FUNCTION_BLOCK FB_Heating_System_Manager
  VAR_INPUT
    VI_System_Mode : E_System_Operating_Mode;
    VI_System_Time_MS : UDINT;
    VI_Current_TOD : TOD;
    VI_IsActivePLC : BOOL;
    VI_Outdoor_Temp : REAL;
    VI_Config : ST_Heating_Config;
    VI_Tariff : ST_Tariff_Config;
    VI_Current_Hour : UINT;
    VI_Boiler_Stop : BOOL;
    VI_DHW_Heating_Demand : BOOL;
    VI_DHW_Target_Temp : REAL;
    VI_Current_Scenario : E_SCENARIO_TYPE;
    VI_Emergency_Stop : BOOL;
    VI_Gas_Safety_Stop : BOOL;
    VI_Boiler_Error_Status : ARRAY[1..GVL_CONSTANTS.C_MAX_BOILERS] OF BOOL;
    VI_Boiler_OT_Online : ARRAY[1..GVL_CONSTANTS.C_MAX_BOILERS] OF BOOL;
    VI_Boiler_Modulation : ARRAY[1..GVL_CONSTANTS.C_MAX_BOILERS] OF REAL;
  END_VAR
  VAR_OUTPUT
    VO_Manifold_Valves : ARRAY[1..GVL_CONSTANTS.C_MAX_MANIFOLDS] OF REAL;
    VO_Manifold_Pumps : ARRAY[1..GVL_CONSTANTS.C_MAX_MANIFOLDS] OF BOOL;
    VO_Zone_Valves : ARRAY[1..GVL_CONSTANTS.C_MAX_HEATING_CIRCUITS] OF BOOL;
    VO_Boiler_OT_Enable : ARRAY[1..GVL_CONSTANTS.C_MAX_BOILERS] OF BOOL;
    VO_Boiler_OT_Setpoint : ARRAY[1..GVL_CONSTANTS.C_MAX_BOILERS] OF REAL;
    VO_Backup_Circulation_Pump : BOOL;
    VO_Electric_Heater_Enable : BOOL;
    VO_Freeze_Risk_Status : BOOL;
    VO_Status : ARRAY[1..GVL_CONSTANTS.C_MAX_MANIFOLDS] OF ST_Manifold_Status;
    VO_Boiler_Status : ARRAY[1..GVL_CONSTANTS.C_MAX_BOILERS] OF ST_Boiler_Status;
  END_VAR
  VAR_IN_OUT
    VI_Floor_Temps : ARRAY[1..GVL_CONSTANTS.C_MAX_HEATING_CIRCUITS] OF REAL;
    VI_Room_Temps : ARRAY[1..GVL_CONSTANTS.C_MAX_CLIMATE_ZONES] OF REAL;
    VI_Manifold_Pressures : ARRAY[1..GVL_CONSTANTS.C_MAX_MANIFOLDS] OF REAL;
    VI_Manifold_Currents : ARRAY[1..GVL_CONSTANTS.C_MAX_MANIFOLDS] OF REAL;
    VI_Manifold_Temps_Supply : ARRAY[1..GVL_CONSTANTS.C_MAX_MANIFOLDS] OF REAL;
    VI_Manifold_Temps_Return : ARRAY[1..GVL_CONSTANTS.C_MAX_MANIFOLDS] OF REAL;
    VI_Boiler_Flame_Status : ARRAY[1..GVL_CONSTANTS.C_MAX_BOILERS] OF BOOL;
    VI_Zone_Configs : ARRAY[1..GVL_CONSTANTS.C_MAX_HEATING_CIRCUITS] OF ST_FloorHeating_Circuit_Config;
    VI_Rule_Actions : ARRAY[1..GVL_CONSTANTS.C_MAX_RULES] OF ST_Rule_Action;
    VI_IO_Modules_Online : ARRAY[1..GVL_CONSTANTS.C_MAX_MODULES] OF BOOL;
    VI_Scenario_Configs : ARRAY[1..GVL_CONSTANTS.C_MAX_SCENARIOS] OF ST_Scenario_Config;
    VI_Manifold_End_Switches : ARRAY[1..GVL_CONSTANTS.C_MAX_MANIFOLDS] OF BOOL;
    VI_Valve_Test_Config : ARRAY[1..GVL_CONSTANTS.C_MAX_MANIFOLDS] OF ST_Valve_Test_Config;
  END_VAR
  VAR
    fbHeatingV2Staging : FB_Heating_V2_Staging_DRAFT;
    L_Heating_V2_Command_Shadow : ST_Heating_Command_V2;
    L_Heating_V2_State_Shadow : ST_Heating_State_V2;
    L_Heating_V2_Shadow_Diff_Found : BOOL;
    L_Heating_V2_Switch_Enabled : BOOL;
    L_Heating_V2_Path_Ready : BOOL;
    L_Heating_Using_Legacy_Fallback : BOOL;
    L_PID_Valves : ARRAY[1..GVL_CONSTANTS.C_MAX_MANIFOLDS] OF FB_PID_Controller;
    L_PID_Timer : ARRAY[1..GVL_CONSTANTS.C_MAX_MANIFOLDS] OF FB_System_Timer;
    L_Floor_Controllers : ARRAY[1..GVL_CONSTANTS.C_MAX_HEATING_CIRCUITS] OF FB_FloorHeating_Controller;
    L_Last_Boiler_Rotation : UDINT;
    L_Lead_Boiler : BYTE := 1;
    L_i : INT;
    L_Zone_Config : ST_FloorHeating_Circuit_Config;
    L_j : INT;
    L_Target_Supply_Temp : REAL;
    L_Demand_Power : REAL;
    L_Any_Zone_Active : ARRAY[1..GVL_CONSTANTS.C_MAX_MANIFOLDS] OF BOOL;
    L_Current_Temp : REAL;
    L_Sensor_Error : BOOL;
    L_Prev_Scenario : E_SCENARIO_TYPE;
    L_Scenario_Adjust : REAL;
    L_Target_Scenario_Adjust : REAL;
    L_Transition_Temp : FB_Scenario_Transition_Controller;
    L_Overheat_Timer : ARRAY[1..GVL_CONSTANTS.C_MAX_HEATING_CIRCUITS] OF FB_System_Timer;
    L_Pump_Run_Timer : ARRAY[1..GVL_CONSTANTS.C_MAX_MANIFOLDS] OF FB_System_Timer;
    L_Pump_Pause_Timer : ARRAY[1..GVL_CONSTANTS.C_MAX_MANIFOLDS] OF FB_System_Timer;
    L_Pump_In_Pause : ARRAY[1..GVL_CONSTANTS.C_MAX_MANIFOLDS] OF BOOL;
    L_Last_Scan_Time : UDINT;
    L_Scan_Time_Init : BOOL := FALSE;
    L_Lifespan_S : REAL := 50000.0 * 3600.0;
    L_Delta_MS : UDINT;
    L_Pump_Diag : ARRAY[1..GVL_CONSTANTS.C_MAX_MANIFOLDS] OF FB_Device_Predictive_Diag;
    L_Boiler_Life : ARRAY[1..GVL_CONSTANTS.C_MAX_BOILERS] OF FB_Lifetime_Predictor;
    fbFloorTempValidator : ARRAY[1..GVL_CONSTANTS.C_MAX_HEATING_CIRCUITS] OF FB_Analog_Validator;
    fbRoomTempValidator : ARRAY[1..GVL_CONSTANTS.C_MAX_CLIMATE_ZONES] OF FB_Analog_Validator;
    fbValveTestManager : FB_Valve_Test_Manager;
    fbBoilerCascade : FB_Boiler_Cascade_Manager;
    fbBoilerOpenTherm : FB_Boiler_OpenTherm_Interface;
    L_IO_Failsafe_Active : BOOL;
    L_Freeze_Mode_Active : BOOL;
    L_Freeze_Target_Supply : REAL;
    L_Delta_T : REAL;
    L_Min_Supply_Temp : REAL;
    L_Boiler_OT_Command_Valid : ARRAY[1..GVL_CONSTANTS.C_MAX_BOILERS] OF BOOL;
    L_Boiler_Request_Enable : ARRAY[1..GVL_CONSTANTS.C_MAX_BOILERS] OF BOOL;
    L_Boiler_Request_Setpoint : ARRAY[1..GVL_CONSTANTS.C_MAX_BOILERS] OF REAL;
    L_Policy_Normal : BOOL;
    L_Policy_Safe_Stop : BOOL;
    L_Policy_Degraded : BOOL;
    L_Policy_Freeze_Protection : BOOL;
    L_Any_Sensor_Error : BOOL;
    L_Any_Subsystem_Degraded : BOOL;
  END_VAR

      // ==============================================================================
// Блок управления системой отопления (Heating System Manager)
// Назначение:
// - Управление контурами теплого пола (открытие/закрытие клапанов).
// - Управление насосами коллекторов и смесительными узлами.
// - Управление каскадом котлов (ротация, расчет ресурса).
// - Защита от перегрева и замерзания.
// - Интеграция с Rule Engine.
// ==============================================================================





// ========================================
// Heating policy layer (phase2)
// ========================================
L_Policy_Normal := (VI_System_Mode = E_System_Operating_Mode.MODE_NORMAL);
L_Policy_Safe_Stop := (VI_System_Mode = E_System_Operating_Mode.MODE_SAFE_STOP);
L_Policy_Degraded := (VI_System_Mode = E_System_Operating_Mode.MODE_DEGRADED);
L_Policy_Freeze_Protection := (VI_System_Mode = E_System_Operating_Mode.MODE_FREEZE_PROTECTION);

// ========================================
// Heating freeze policy activation
// ========================================
IF L_Policy_Freeze_Protection THEN
    L_Freeze_Mode_Active := TRUE;
END_IF;

// 0. Агрегация деградации для system mode
GVL_STATE.G_Heating_IO_Fault := FALSE;
GVL_STATE.G_Heating_Sensor_Fault := FALSE;
GVL_STATE.G_Heating_Subsystem_Degraded := FALSE;
L_Any_Sensor_Error := FALSE;
L_Any_Subsystem_Degraded := FALSE;
L_Heating_V2_Shadow_Diff_Found := FALSE;
L_Heating_V2_Switch_Enabled := TRUE;
L_Heating_V2_Path_Ready := FALSE;
L_Heating_Using_Legacy_Fallback := TRUE;

// 0. Аварийный стоп от подсистемы безопасности
VO_Backup_Circulation_Pump := FALSE;
VO_Electric_Heater_Enable := FALSE;
VO_Freeze_Risk_Status := FALSE;

IF VI_Gas_Safety_Stop THEN
    L_Freeze_Mode_Active := (VI_Outdoor_Temp < -5.0);
    FOR L_i := 1 TO GVL_CONSTANTS.C_MAX_HEATING_CIRCUITS DO
        IF VI_Floor_Temps[L_i] < 7.0 THEN
            L_Freeze_Mode_Active := TRUE;
        END_IF;
        VO_Zone_Valves[L_i] := FALSE;
    END_FOR;

    FOR L_i := 1 TO GVL_CONSTANTS.C_MAX_MANIFOLDS DO
        VO_Manifold_Pumps[L_i] := FALSE;
        VO_Manifold_Valves[L_i] := 0.0;
    END_FOR;

    FOR L_i := 1 TO GVL_CONSTANTS.C_MAX_BOILERS DO
        VO_Boiler_OT_Enable[L_i] := FALSE;
        VO_Boiler_OT_Setpoint[L_i] := 0.0;
        VO_Boiler_Status[L_i].Warning := FALSE;
        VO_Boiler_Status[L_i].Error := TRUE;
    END_FOR;

    IF L_Freeze_Mode_Active THEN
        VO_Backup_Circulation_Pump := TRUE;
        L_Freeze_Target_Supply := LIMIT(20.0, VI_Config.Freeze_Threshold + 2.0, 35.0);
        L_Min_Supply_Temp := 1000.0;
        FOR L_i := 1 TO GVL_CONSTANTS.C_MAX_MANIFOLDS DO
            IF VI_Manifold_Temps_Supply[L_i] < L_Min_Supply_Temp THEN
                L_Min_Supply_Temp := VI_Manifold_Temps_Supply[L_i];
            END_IF;
        END_FOR;
        IF L_Min_Supply_Temp > 900.0 THEN
            L_Min_Supply_Temp := 0.0;
        END_IF;

        IF L_Min_Supply_Temp < (L_Freeze_Target_Supply - 1.0) THEN
            VO_Electric_Heater_Enable := TRUE;
        ELSIF L_Min_Supply_Temp > (L_Freeze_Target_Supply + 1.0) THEN
            VO_Electric_Heater_Enable := FALSE;
        END_IF;

        // При защёлкнутой газовой аварии оператор должен видеть, что система живёт в деградированном anti-freeze режиме.
        VO_Freeze_Risk_Status := TRUE;
    END_IF;

    RETURN;
END_IF;

IF VI_Emergency_Stop OR L_Policy_Safe_Stop THEN
    FOR L_i := 1 TO GVL_CONSTANTS.C_MAX_HEATING_CIRCUITS DO
        VO_Zone_Valves[L_i] := FALSE;
    END_FOR;

    FOR L_i := 1 TO GVL_CONSTANTS.C_MAX_MANIFOLDS DO
        VO_Manifold_Pumps[L_i] := FALSE;
        VO_Manifold_Valves[L_i] := 0.0;
    END_FOR;

    FOR L_i := 1 TO GVL_CONSTANTS.C_MAX_BOILERS DO
        VO_Boiler_OT_Enable[L_i] := FALSE;
        VO_Boiler_OT_Setpoint[L_i] := 0.0;
        VO_Boiler_Status[L_i].Warning := FALSE;
        VO_Boiler_Status[L_i].Error := TRUE;
    END_FOR;

    RETURN;
END_IF;

// 1. Проверка связи с модулями ввода-вывода (ТЗ 2.0)
L_IO_Failsafe_Active := FALSE;
FOR L_i := 1 TO GVL_CONSTANTS.C_MAX_MODULES DO
    IF NOT VI_IO_Modules_Online[L_i] THEN
        L_IO_Failsafe_Active := TRUE;
        GVL_STATE.G_Heating_IO_Fault := TRUE;
GVL_STATE.G_Heating_Subsystem_Degraded := TRUE;
        EXIT;
    END_IF;
END_FOR;

IF L_IO_Failsafe_Active THEN
    // Fail-safe: закрываем зональные клапаны, чтобы не разгонять неконтролируемые контуры,
    // но при риске замерзания сохраняем минимальную циркуляцию и минимальную теплогенерацию.
    L_Freeze_Mode_Active := (VI_Outdoor_Temp < -5.0);

    FOR L_j := 1 TO GVL_CONSTANTS.C_MAX_HEATING_CIRCUITS DO
        IF VI_Floor_Temps[L_j] < 7.0 THEN
            L_Freeze_Mode_Active := TRUE;
        END_IF;
        VO_Zone_Valves[L_j] := FALSE;
    END_FOR;

    IF L_Freeze_Mode_Active THEN
        L_Freeze_Target_Supply := LIMIT(20.0, VI_Config.Freeze_Threshold + 2.0, 35.0);
    ELSE
        L_Freeze_Target_Supply := 0.0;
    END_IF;

    FOR L_j := 1 TO GVL_CONSTANTS.C_MAX_MANIFOLDS DO
        IF L_Freeze_Mode_Active THEN
            VO_Manifold_Pumps[L_j] := TRUE;
            VO_Manifold_Valves[L_j] := 35.0;
        ELSE
            VO_Manifold_Pumps[L_j] := FALSE;
            VO_Manifold_Valves[L_j] := 0.0;
        END_IF;
    END_FOR;

    // В аварийном I/O режиме напрямую формируем только legacy request-мirror.
    // Реальные физические команды всё равно будут интерпретированы transport-слоем выше по архитектуре.
    FOR L_j := 1 TO GVL_CONSTANTS.C_MAX_BOILERS DO
        VO_Boiler_OT_Enable[L_j] := FALSE;
        VO_Boiler_OT_Setpoint[L_j] := 0.0;
    END_FOR;

    IF L_Freeze_Mode_Active THEN
        // В fail-safe используем только ведущий аварийный вариант: котёл №1 на минимальной уставке.
        IF VI_Boiler_OT_Online[1] AND NOT VI_Boiler_Error_Status[1] THEN
            VO_Boiler_OT_Enable[1] := TRUE;
            VO_Boiler_OT_Setpoint[1] := L_Freeze_Target_Supply;
        END_IF;
    END_IF;

    RETURN;
END_IF;

// 2. Расчет целевой температуры подачи теплоносителя (Погодозависимая автоматика ТЗ 2.3)
L_Target_Supply_Temp := 35.0; // Базовая уставка
IF VI_Config.Weather_Comp_Enabled AND VI_Outdoor_Temp < 15.0 THEN
    // Коррекция по уличному датчику с использованием коэффициента кривой
    L_Target_Supply_Temp := L_Target_Supply_Temp + (15.0 - VI_Outdoor_Temp) * VI_Config.Weather_Coef;
END_IF;
L_Target_Supply_Temp := LIMIT(20.0, L_Target_Supply_Temp, 45.0); // Ограничение диапазона для теплого пола

IF L_Policy_Degraded THEN
    IF L_Target_Supply_Temp > 35.0 THEN
        L_Target_Supply_Temp := 35.0;
    END_IF;
END_IF;

// Плавный переход уставки по сценарию
IF VI_Current_Scenario >= 1 AND VI_Current_Scenario <= GVL_CONSTANTS.C_MAX_SCENARIOS THEN
    L_Target_Scenario_Adjust := VI_Scenario_Configs[VI_Current_Scenario].floor_heating_adjust_celsius;
ELSE
    L_Target_Scenario_Adjust := 0.0;
END_IF;

IF VI_Current_Scenario <> L_Prev_Scenario THEN
    L_Transition_Temp(
        VI_System_Time := VI_System_Time_MS,
        VI_Start_Time := VI_System_Time_MS,
        VI_Duration := 300000, // 5 минут на плавное изменение температуры
        VI_Start_Value := L_Scenario_Adjust,
        VI_End_Value := L_Target_Scenario_Adjust
    );
    L_Prev_Scenario := VI_Current_Scenario;
ELSE
    L_Transition_Temp(
        VI_System_Time := VI_System_Time_MS,
        VI_Start_Time := L_Transition_Temp.VI_Start_Time,
        VI_Duration := L_Transition_Temp.VI_Duration,
        VI_Start_Value := L_Transition_Temp.VI_Start_Value,
        VI_End_Value := L_Target_Scenario_Adjust
    );
END_IF;
L_Scenario_Adjust := L_Transition_Temp.VO_Current_Value;

// ТЗ 2.4: Защита от замерзания по температуре пола < 7°C или наружной < -5°C
L_Freeze_Mode_Active := L_Policy_Freeze_Protection OR (VI_Outdoor_Temp < -5.0);
IF NOT L_Freeze_Mode_Active THEN
    FOR L_i := 1 TO GVL_CONSTANTS.C_MAX_HEATING_CIRCUITS DO
        IF VI_Floor_Temps[L_i] < 7.0 THEN
            L_Freeze_Mode_Active := TRUE;
            EXIT;
        END_IF;
    END_FOR;
END_IF;

IF L_Freeze_Mode_Active THEN
    L_Freeze_Target_Supply := LIMIT(20.0, VI_Config.Freeze_Threshold + 2.0, 45.0);
    IF L_Target_Supply_Temp < L_Freeze_Target_Supply THEN
        L_Target_Supply_Temp := L_Freeze_Target_Supply;
    END_IF;
END_IF;

// 2. Индивидуальное управление зонами отопления (ТЗ 1.1, 2.5)
FOR L_i := 1 TO GVL_CONSTANTS.C_MAX_HEATING_CIRCUITS DO
    fbFloorTempValidator[L_i](
        VI_Value := VI_Floor_Temps[L_i],
        VI_Min_Valid := -40.0,
        VI_Max_Valid := 120.0,
        VI_Fallback_Mode := 0
    );
    
    L_Climate_Zone_ID := VI_Zone_Configs[L_i].zone;
    IF L_Climate_Zone_ID >= 1 AND L_Climate_Zone_ID <= GVL_CONSTANTS.C_MAX_CLIMATE_ZONES THEN
        fbRoomTempValidator[L_Climate_Zone_ID](
        VI_Value := VI_Room_Temps[L_Climate_Zone_ID],
        VI_Min_Valid := -40.0,
        VI_Max_Valid := 120.0,
        VI_Fallback_Mode := 0
        );
    END_IF;

    // Контроль перегрева стяжки (защита напольного покрытия)
    L_Overheat_Timer[L_i](IN := fbFloorTempValidator[L_i].VO_Value > VI_Config.Overheat_Threshold, PT := T#60s, VI_System_Time_MS := VI_System_Time_MS);
    
    // Выбор датчика температуры с автоматическим переключением при неисправности
    L_Current_Temp := 0.0;
    L_Sensor_Error := FALSE;
    
    IF VI_Zone_Configs[L_i].control_type = 1 OR VI_Zone_Configs[L_i].control_type = 2 THEN
        // Основной: по воздуху
        IF NOT fbRoomTempValidator[L_Climate_Zone_ID].VO_Error THEN
            L_Current_Temp := fbRoomTempValidator[L_Climate_Zone_ID].VO_Value;
        ELSIF NOT fbFloorTempValidator[L_i].VO_Error THEN
            L_Current_Temp := fbFloorTempValidator[L_i].VO_Value; // Резервный: по полу
        ELSE
            L_Sensor_Error := TRUE;
        END_IF;
    ELSE
        // Основной: по полу
        IF NOT fbFloorTempValidator[L_i].VO_Error THEN
            L_Current_Temp := fbFloorTempValidator[L_i].VO_Value;
        ELSIF NOT fbRoomTempValidator[L_Climate_Zone_ID].VO_Error THEN
            L_Current_Temp := fbRoomTempValidator[L_Climate_Zone_ID].VO_Value; // Резервный: по воздуху
        ELSE
            L_Sensor_Error := TRUE;
        END_IF;
    END_IF;

    IF L_Sensor_Error THEN
        L_Any_Sensor_Error := TRUE;
        VO_Zone_Valves[L_i] := FALSE; // Безопасное состояние при ошибке обоих датчиков
    ELSE
        // ПИД-регулирование и ШИМ для каждой зоны
        // Применяем плавную корректировку уставки от сценария
        L_Zone_Config := VI_Zone_Configs[L_i];
        L_Zone_Config.design_temp := L_Zone_Config.design_temp + L_Scenario_Adjust;
        L_Floor_Controllers[L_i](
            VI_Current_Temp := L_Current_Temp,
            VI_Config := L_Zone_Config,
            VI_Tariff := VI_Tariff,
            VI_Current_Hour := VI_Current_Hour,
            VI_IsActivePLC := VI_IsActivePLC,
            VI_System_Time_MS := VI_System_Time_MS,
            VO_Valve_Bool => VO_Zone_Valves[L_i]
        );
    END_IF;
    
    // Принудительное закрытие клапана при перегреве пола (ТЗ 2.5)
    IF L_Overheat_Timer[L_i].Q THEN
        VO_Zone_Valves[L_i] := FALSE;
    END_IF;
    
    // Обработка действий от Rule Engine (ТЗ 13.0)
    FOR L_j := 1 TO GVL_CONSTANTS.C_MAX_RULES DO
        IF VI_Rule_Actions[L_j].Active AND VI_Rule_Actions[L_j].Target_ID = L_i THEN
            IF VI_Rule_Actions[L_j].Action_Type = E_Rule_Action_Type.ACTION_SET_FLOOR_HEATING THEN
                VO_Zone_Valves[L_i] := (VI_Rule_Actions[L_j].Value > 0.5);
            END_IF;
        END_IF;
    END_FOR;
END_FOR;

GVL_STATE.G_Heating_Sensor_Fault := L_Any_Sensor_Error;

// 3. Определение потребности в работе коллекторных насосов
FOR L_i := 1 TO GVL_CONSTANTS.C_MAX_MANIFOLDS DO
    L_Any_Zone_Active[L_i] := FALSE;
END_FOR;

FOR L_i := 1 TO GVL_CONSTANTS.C_MAX_HEATING_CIRCUITS DO
    IF VO_Zone_Valves[L_i] THEN
        L_j := VI_Zone_Configs[L_i].manifold_id;
        IF L_j >= 1 AND L_j <= GVL_CONSTANTS.C_MAX_MANIFOLDS THEN
            L_Any_Zone_Active[L_j] := TRUE;
        END_IF;
    END_IF;
END_FOR;

// 4. Управление смесительными узлами коллекторов (ТЗ 2.6, 12.2)
FOR L_i := 1 TO GVL_CONSTANTS.C_MAX_MANIFOLDS DO
    // ПИД-регулирование трехходового клапана для поддержания стабильной температуры подачи
    // Вызываем ПИД регулятор каждую секунду
    L_PID_Timer[L_i](IN := TRUE, PT := T#1s, VI_System_Time_MS := VI_System_Time_MS);
    IF L_PID_Timer[L_i].Q THEN
        L_PID_Timer[L_i](IN := FALSE, PT := T#1s, VI_System_Time_MS := VI_System_Time_MS); // Сброс таймера
        L_PID_Timer[L_i](IN := TRUE, PT := T#1s, VI_System_Time_MS := VI_System_Time_MS); // Перезапуск
        
        L_PID_Valves[L_i](
            VI_SetPoint := L_Target_Supply_Temp,
            VI_ProcessValue := VI_Manifold_Temps_Supply[L_i],
            VI_Kp := 2.0, VI_Tn := 120.0, VI_Tv := 0.0,
            VI_Y_Min := 0.0, VI_Y_Max := 100.0, VI_Cycle_Time_S := 1.0,
            VO_Output => VO_Manifold_Valves[L_i]
        );
    END_IF;

    // ТЗ 2.6: Реализация обязательной паузы насоса (защита от закисания и перегрева при 72ч работе)
    L_Pump_Run_Timer[L_i](IN := VO_Manifold_Pumps[L_i] AND NOT L_Pump_In_Pause[L_i], PT := T#72h, VI_System_Time_MS := VI_System_Time_MS);
    IF L_Pump_Run_Timer[L_i].Q THEN L_Pump_In_Pause[L_i] := TRUE; END_IF;
    
    L_Pump_Pause_Timer[L_i](IN := L_Pump_In_Pause[L_i], PT := T#1h, VI_System_Time_MS := VI_System_Time_MS);
    IF L_Pump_Pause_Timer[L_i].Q THEN L_Pump_In_Pause[L_i] := FALSE; END_IF;

    // Включение насоса при наличии запроса от зон и отсутствии сервисной паузы
    // Приоритет ГВС: если есть запрос от ГВС, отключаем насосы отопления и закрываем клапаны
    IF VI_DHW_Heating_Demand THEN
        VO_Manifold_Pumps[L_i] := FALSE;
        VO_Manifold_Valves[L_i] := 0.0; // Принудительно закрываем смесительный клапан
    ELSE
        VO_Manifold_Pumps[L_i] := VI_IsActivePLC AND L_Any_Zone_Active[L_i] AND NOT L_Pump_In_Pause[L_i];
    END_IF;

    // Защита от замерзания системы (ТЗ 2.4)
        IF L_Freeze_Mode_Active THEN
            VO_Manifold_Pumps[L_i] := TRUE;
            IF VO_Manifold_Valves[L_i] < 35.0 THEN
                VO_Manifold_Valves[L_i] := 35.0;
            END_IF;
        END_IF;

        // Сбор диагностических данных для визуализации на HMI
    VO_Status[L_i].Pump_On := VO_Manifold_Pumps[L_i];
    VO_Status[L_i].Pump_Current := VI_Manifold_Currents[L_i];
    VO_Status[L_i].Pressure := VI_Manifold_Pressures[L_i];
    VO_Status[L_i].Temp_Supply := VI_Manifold_Temps_Supply[L_i];
    VO_Status[L_i].Temp_Return := VI_Manifold_Temps_Return[L_i];
    VO_Status[L_i].Valve_Pos := VO_Manifold_Valves[L_i];
    
    // Предиктивная диагностика насоса
    L_Pump_Diag[L_i](
        VI_Current_Value := VI_Manifold_Currents[L_i],
        VI_Nominal_Value := 0.55, // Номинальный ток насоса по ТЗ: середина диапазона 0.3..0.8 А
        VI_Is_Running := VO_Manifold_Pumps[L_i],
        VI_Reset_Stats := FALSE,
        VI_System_Time_MS := VI_System_Time_MS,
        VIO_Health_Data := VO_Status[L_i].Health
    );
    
    // Автоматический контроль рабочих параметров (ток / давление / ΔT)
        IF VO_Manifold_Pumps[L_i] THEN
            L_Delta_T := VI_Manifold_Temps_Supply[L_i] - VI_Manifold_Temps_Return[L_i];

            // Контроль тока насоса:
            // Приоритет ошибок:
            // 1. Насос/ток
            // 2. Давление
            // 3. ΔT
            VO_Status[L_i].Error := FALSE;
            VO_Status[L_i].Error_ID := 0;

            IF VI_Manifold_Currents[L_i] <= 0.01 THEN
                VO_Status[L_i].Error := TRUE;
                VO_Status[L_i].Error_ID := GVL_CONFIG.ERR_PUMP_NO_CURRENT;
            ELSIF VI_Manifold_Currents[L_i] < 0.3 THEN
                VO_Status[L_i].Error := TRUE;
                VO_Status[L_i].Error_ID := GVL_CONFIG.ERR_PUMP_UNDERCURRENT;
            ELSIF VI_Manifold_Currents[L_i] > 1.5 THEN
                VO_Status[L_i].Error := TRUE;
                VO_Status[L_i].Error_ID := GVL_CONFIG.ERR_PUMP_OVERCURRENT;
            END_IF;

            // Проверка давления в системе (норма 1.5 - 2.5 бар)
            IF (NOT VO_Status[L_i].Error) AND (VI_Manifold_Pressures[L_i] < 1.5 OR VI_Manifold_Pressures[L_i] > 2.5) THEN
                VO_Status[L_i].Error := TRUE;
                VO_Status[L_i].Error_ID := GVL_CONFIG.ERR_PRESSURE_OUT_OF_RANGE;
            END_IF;

            // Проверка эффективности теплообмена (ΔT 5..10°C норма)
            IF NOT VO_Status[L_i].Error THEN
                IF L_Delta_T < 5.0 THEN
                    VO_Status[L_i].Error := TRUE;
                    VO_Status[L_i].Error_ID := GVL_CONFIG.ERR_DELTA_T_LOW;
                ELSIF L_Delta_T > 10.0 THEN
                    VO_Status[L_i].Error := TRUE;
                    VO_Status[L_i].Error_ID := GVL_CONFIG.ERR_DELTA_T_HIGH;
                END_IF;
            END_IF;
        END_IF;

        // ТЗ 12.2: Еженедельное тестирование запорной арматуры (предотвращение закисания)
    // Выполняется менеджером fbValveTestManager
END_FOR;

fbValveTestManager(
    VI_System_Time_MS := VI_System_Time_MS,
    VI_IsActivePLC := VI_IsActivePLC,
    VI_Valve_Currents := VI_Manifold_Currents,
    VI_Valve_End_Switches := VI_Manifold_End_Switches,
    VI_Config := VI_Valve_Test_Config
);

IF fbValveTestManager.VO_Test_Active THEN
    L_i := fbValveTestManager.VO_Current_Valve;
    IF L_i >= 1 AND L_i <= GVL_CONSTANTS.C_MAX_MANIFOLDS THEN
        IF fbValveTestManager.VO_Valve_Cmd[L_i] THEN
            VO_Manifold_Valves[L_i] := 100.0;
        ELSE
            VO_Manifold_Valves[L_i] := 0.0;
        END_IF;
        VO_Manifold_Pumps[L_i] := FALSE; // Отключаем насос при тестировании клапана
    END_IF;
END_IF;

// 5. Управление каскадом котлов (ТЗ 2.8, OpenTherm-only, без legacy mirror)
L_Demand_Power := 0.0;
FOR L_i := 1 TO GVL_CONSTANTS.C_MAX_MANIFOLDS DO
    IF VO_Manifold_Pumps[L_i] THEN
        L_Demand_Power := L_Demand_Power + VO_Manifold_Valves[L_i];
    END_IF;
END_FOR;

// В режиме антизамерзания обеспечиваем минимальный запрос тепла
IF L_Freeze_Mode_Active AND L_Demand_Power < 20.0 THEN
    L_Demand_Power := 20.0;
END_IF;

IF L_Policy_Degraded THEN
    IF L_Demand_Power > 60.0 THEN
        L_Demand_Power := 60.0;
    END_IF;
END_IF;

fbBoilerCascade(
    VI_Enable := VI_IsActivePLC AND ((L_Demand_Power > GVL_CONSTANTS.C_BOILER_CASCADE_MIN_DEMAND) OR L_Freeze_Mode_Active),
    VI_System_Time_MS := VI_System_Time_MS,
    VI_Boiler_Stop := FALSE,
    VI_DHW_Heating_Demand := VI_DHW_Heating_Demand,
    VI_DHW_Target_Temp := VI_DHW_Target_Temp,
    VI_Target_Supply_Temp := L_Target_Supply_Temp,
    VI_Demand_Power := L_Demand_Power,
    VI_Boiler_Flame_Status := VI_Boiler_Flame_Status,
    VI_Boiler_Error_Status := VI_Boiler_Error_Status,
    VI_Boiler_OT_Online := VI_Boiler_OT_Online,
    VI_Boiler_Modulation := VI_Boiler_Modulation,
    VO_Boiler_Enable => L_Boiler_Request_Enable,
    VO_Boiler_Setpoint => L_Boiler_Request_Setpoint,
    VO_Lead_Boiler => L_Lead_Boiler
);



// ========================================
// OT availability enforcement (no fallback)
// ========================================
FOR L_i := 1 TO GVL_CONSTANTS.C_MAX_BOILERS DO
    IF NOT VI_Boiler_OT_Online[L_i] OR VI_Boiler_Error_Status[L_i] THEN
        L_Boiler_Request_Enable[L_i] := FALSE;
        L_Boiler_Request_Setpoint[L_i] := 0.0;
    END_IF;
END_FOR;

fbBoilerOpenTherm(
    VI_Enable := L_Boiler_Request_Enable,
    VI_Setpoint := L_Boiler_Request_Setpoint,
    VI_OT_Online := VI_Boiler_OT_Online,
    VI_OT_Error := VI_Boiler_Error_Status,
    VO_OT_Enable => VO_Boiler_OT_Enable,
    VO_OT_Setpoint => VO_Boiler_OT_Setpoint,
    VO_OT_Command_Valid => L_Boiler_OT_Command_Valid
);


// ========================================
// Boiler status normalization
// ========================================
FOR L_i := 1 TO GVL_CONSTANTS.C_MAX_BOILERS DO
    // Базовый сброс диагностических флагов котла
    VO_Boiler_Status[L_i].Active := L_Boiler_Request_Enable[L_i];
    VO_Boiler_Status[L_i].Warning := FALSE;
    VO_Boiler_Status[L_i].Error := FALSE;

    // Приоритет причин:
    // 1. Нет канала OpenTherm
    // 2. Котёл вернул ошибку
    // 3. Есть запрос, но нет пламени
    IF NOT VI_Boiler_OT_Online[L_i] THEN
        VO_Boiler_Status[L_i].Error := TRUE;
        VO_Boiler_Status[L_i].Error_ID := GVL_CONFIG.ERR_BOILER_OFFLINE;
        L_Any_Subsystem_Degraded := TRUE;
    ELSIF VI_Boiler_Error_Status[L_i] THEN
        VO_Boiler_Status[L_i].Error := TRUE;
        VO_Boiler_Status[L_i].Error_ID := GVL_CONFIG.ERR_BOILER_GENERAL_FAULT;
        L_Any_Subsystem_Degraded := TRUE;
    ELSIF L_Boiler_Request_Enable[L_i] AND NOT VI_Boiler_Flame_Status[L_i] THEN
        VO_Boiler_Status[L_i].Warning := TRUE;
        VO_Boiler_Status[L_i].Error_ID := GVL_CONFIG.ERR_BOILER_NO_FLAME;
        L_Any_Subsystem_Degraded := TRUE;
    ELSE
        VO_Boiler_Status[L_i].Error_ID := 0;
    END_IF;
END_FOR;

// Расчет наработки и остаточного ресурса котлов (ТЗ 2.8)
IF NOT L_Scan_Time_Init THEN
    L_Last_Scan_Time := VI_System_Time_MS;
    L_Scan_Time_Init := TRUE;
END_IF;

L_Delta_MS := F_TimeDiff(VI_System_Time_MS, L_Last_Scan_Time);
IF L_Delta_MS > 1000 THEN
    L_Delta_MS := 1000; // Ограничение дельты для предотвращения скачков после перезагрузки
END_IF;

L_Last_Scan_Time := VI_System_Time_MS;

FOR L_i := 1 TO GVL_CONSTANTS.C_MAX_BOILERS DO
    VO_Boiler_Status[L_i].Work_Seconds := GVL_Retain.G_Boiler_Work_Seconds[L_i];
    
    IF VI_Boiler_Flame_Status[L_i] THEN
        GVL_Retain.G_Boiler_Accumulated_MS[L_i] := GVL_Retain.G_Boiler_Accumulated_MS[L_i] + L_Delta_MS;
        IF GVL_Retain.G_Boiler_Accumulated_MS[L_i] >= GVL_CONSTANTS.C_MS_IN_SECOND THEN
            GVL_Retain.G_Boiler_Work_Seconds[L_i] := GVL_Retain.G_Boiler_Work_Seconds[L_i] + (GVL_Retain.G_Boiler_Accumulated_MS[L_i] / 1000);
            GVL_Retain.G_Boiler_Accumulated_MS[L_i] := GVL_Retain.G_Boiler_Accumulated_MS[L_i] MOD 1000;
            
            // Защита от переполнения (сброс при достижении ~136 лет)
            IF GVL_Retain.G_Boiler_Work_Seconds[L_i] > 4000000000 THEN
                GVL_Retain.G_Boiler_Work_Seconds[L_i] := 0;
            END_IF;
            
            VO_Boiler_Status[L_i].Work_Seconds := GVL_Retain.G_Boiler_Work_Seconds[L_i];
        END_IF;
    END_IF;
    
    VO_Boiler_Status[L_i].Work_Hours := TO_REAL(VO_Boiler_Status[L_i].Work_Seconds) / 3600.0;
    
    L_Boiler_Life[L_i](
        VI_Runtime_Hours := TO_UDINT(VO_Boiler_Status[L_i].Work_Hours),
        VI_Start_Count := 0, // Не считаем пуски для котлов в этой версии
        VI_Nominal_Life := 50000 // 50,000 часов
    );
    VO_Boiler_Status[L_i].Resource_Percent := TO_REAL(L_Boiler_Life[L_i].VO_Remaining_Percent);
    VO_Boiler_Status[L_i].Running := VI_Boiler_Flame_Status[L_i];
END_FOR;
GVL_STATE.G_Heating_Subsystem_Degraded := L_Any_Subsystem_Degraded;

// ========================================
// Heating V2 shadow execution (phase2)
// ========================================
fbHeatingV2Staging(
    VI_Zone_ID := 1,
    VI_Enable := TRUE,
    VI_Target_Temp := 22.0,
    VI_Valve_Position_Setpoint := 50.0,
    VI_Pump_Enable := TRUE,

    VI_Is_Active := TRUE,
    VI_Room_Temp := 21.0,
    VI_Supply_Temp := 35.0,
    VI_Return_Temp := 30.0,
    VI_Valve_Position_Actual := 50.0,
    VI_Alarm_Active := FALSE,

    VO_Command_Shadow => L_Heating_V2_Command_Shadow,
    VO_State_Shadow => L_Heating_V2_State_Shadow
);

// Heating V2 shadow validation
IF ABS(VO_Manifold_Valves[1] - L_Heating_V2_Command_Shadow.Valve_Position_Setpoint) > 0.1 THEN
    L_Heating_V2_Shadow_Diff_Found := TRUE;
END_IF;
IF ABS(VI_Room_Temps[1] - L_Heating_V2_State_Shadow.Room_Temp) > 0.1 THEN
    L_Heating_V2_Shadow_Diff_Found := TRUE;
END_IF;
IF ABS(VI_Manifold_Temps_Supply[1] - L_Heating_V2_State_Shadow.Supply_Temp) > 0.1 THEN
    L_Heating_V2_Shadow_Diff_Found := TRUE;
END_IF;

// Guarded Heating V2 enable
IF L_Heating_V2_Switch_Enabled THEN
    IF NOT L_Heating_V2_Shadow_Diff_Found THEN
        L_Heating_V2_Path_Ready := TRUE;
        L_Heating_Using_Legacy_Fallback := FALSE;
    ELSE
        L_Heating_V2_Path_Ready := FALSE;
        L_Heating_Using_Legacy_Fallback := TRUE;
    END_IF;
ELSE
    L_Heating_V2_Path_Ready := FALSE;
    L_Heating_Using_Legacy_Fallback := TRUE;
END_IF;

// >>> BULK_SYNC_ANCHOR: FB_Heating_System_Manager <<<
    
END_FUNCTION_BLOCK

FUNCTION_BLOCK FB_History_Manager
  VAR_INPUT
    VI_System_Time_MS : UDINT;
    VI_Write_Event : BOOL;
    VI_Event : ST_History_Record;
  END_VAR
  VAR_OUTPUT
    VO_Total_Events : UDINT;
  END_VAR
  VAR
    L_Prev_Write_Event : BOOL;
  END_VAR

      IF VI_Write_Event AND NOT L_Prev_Write_Event THEN
    GVL_Retain.G_History_Buffer[GVL_Retain.G_History_Write_Idx] := VI_Event;
    GVL_Retain.G_History_Buffer[GVL_Retain.G_History_Write_Idx].timestamp_ms := VI_System_Time_MS;
    
    GVL_Retain.G_History_Write_Idx := (GVL_Retain.G_History_Write_Idx MOD GVL_CONSTANTS.C_MAX_HISTORY_RECORDS) + 1;
    GVL_Retain.G_History_Total_Events := GVL_Retain.G_History_Total_Events + 1;
END_IF;
L_Prev_Write_Event := VI_Write_Event;

VO_Total_Events := GVL_Retain.G_History_Total_Events;
// >>> BULK_SYNC_ANCHOR: FB_History_Manager <<<
    
END_FUNCTION_BLOCK

FUNCTION_BLOCK FB_IO_Module_Watchdog
  VAR_INPUT
    VI_System_Time_MS : UDINT;
    VI_Module_ID : BYTE;
    VI_Heartbeat_Signal : BOOL;
    VI_Timeout_MS : UDINT := 2000;
  END_VAR
  VAR_OUTPUT
    VO_Module_Online : BOOL;
    VO_Error_Active : BOOL;
  END_VAR
  VAR
    L_Last_Heartbeat_State : BOOL;
    L_Last_Heartbeat_Time : UDINT;
    L_Elapsed_Time : UDINT;
  END_VAR

      // Отслеживание изменения сигнала
IF VI_Heartbeat_Signal <> L_Last_Heartbeat_State THEN
    L_Last_Heartbeat_Time := VI_System_Time_MS;
    L_Last_Heartbeat_State := VI_Heartbeat_Signal;
END_IF;

// Проверка таймаута
L_Elapsed_Time := F_TimeDiff(VI_System_Time_MS, L_Last_Heartbeat_Time);

IF L_Elapsed_Time > VI_Timeout_MS THEN
    VO_Module_Online := FALSE;
    VO_Error_Active := TRUE;
ELSE
    VO_Module_Online := TRUE;
    VO_Error_Active := FALSE;
END_IF;
// >>> BULK_SYNC_ANCHOR: FB_IO_Module_Watchdog <<<
    
END_FUNCTION_BLOCK

FUNCTION_BLOCK FB_Lighting_Blinds_Manager
  VAR_INPUT
    VI_System_Time_MS : UDINT;
    VI_IsActivePLC : BOOL;
    VI_Current_Scenario : E_SCENARIO_TYPE;
    VI_Away_Level : BYTE;
    VI_Simulation_Active : BOOL;
    VI_Is_Night : BOOL;
    VI_System_Mode : E_System_Operating_Mode;
  END_VAR
  VAR_OUTPUT
    VO_Lighting_Levels : ARRAY[1..GVL_CONSTANTS.C_MAX_LIGHTING_ZONES] OF BYTE;
    VO_Blinds_Positions : ARRAY[1..GVL_CONSTANTS.C_MAX_BLINDS] OF BYTE;
    VO_Wet_Zone_Light_Active : ARRAY[1..GVL_CONSTANTS.C_MAX_WET_ZONES] OF BOOL;
  END_VAR
  VAR_IN_OUT
    VI_Manual_Light_Override : ARRAY[1..GVL_CONSTANTS.C_MAX_LIGHTING_ZONES] OF BYTE;
    VI_Manual_Blinds_Override : ARRAY[1..GVL_CONSTANTS.C_MAX_BLINDS] OF BYTE;
    VI_Simulation_Lights : ARRAY[1..GVL_CONSTANTS.C_MAX_LIGHTING_ZONES] OF BOOL;
    VI_Physical_Switches : ARRAY[1..GVL_CONSTANTS.C_MAX_LIGHTING_ZONES] OF BOOL;
    VI_Motion_Sensors : ARRAY[1..GVL_CONSTANTS.C_MAX_LIGHTING_ZONES] OF BOOL;
    VI_Rule_Actions : ARRAY[1..GVL_CONSTANTS.C_MAX_RULES] OF ST_Rule_Action;
    VI_IO_Modules_Online : ARRAY[1..GVL_CONSTANTS.C_MAX_MODULES] OF BOOL;
    VI_Wet_Zone_Map : ARRAY[1..GVL_CONSTANTS.C_MAX_LIGHTING_ZONES] OF BOOL;
    VI_Scenario_Configs : ARRAY[1..GVL_CONSTANTS.C_MAX_SCENARIOS] OF ST_Scenario_Config;
  END_VAR
  VAR
    fbBlindsV2Staging : FB_Blinds_V2_Staging;
    L_Blinds_V2_Command_Shadow : ST_Blinds_Command_V2;
    L_Blinds_V2_State_Shadow : ST_Blinds_State_V2;
    L_Blinds_V2_Shadow_Diff_Found : BOOL;
    L_Blinds_V2_Switch_Enabled : BOOL;
    L_Blinds_V2_Path_Ready : BOOL;
    L_Blinds_Using_Legacy_Fallback : BOOL;
    fbLightingV2Staging : FB_Lighting_V2_Staging;
    L_Lighting_V2_Command_Shadow : ST_Lighting_Command_V2;
    L_Lighting_V2_State_Shadow : ST_Lighting_State_V2;
    L_Lighting_V2_Shadow_Diff_Found : BOOL;
    L_Lighting_V2_Switch_Enabled : BOOL;
    L_Lighting_V2_Path_Ready : BOOL;
    L_Lighting_Using_Legacy_Fallback : BOOL;
    L_i : INT;
    L_j : INT;
    L_Base_Light : BYTE;
    L_Base_Blinds : BYTE;
    L_Target_Base_Light : BYTE;
    L_Target_Base_Blinds : BYTE;
    L_Prev_Scenario : E_SCENARIO_TYPE;
    L_Transition_Light : FB_Scenario_Transition_Controller;
    L_Transition_Blinds : FB_Scenario_Transition_Controller;
    L_Light_States : ARRAY[1..GVL_CONSTANTS.C_MAX_LIGHTING_ZONES] OF BOOL;
    L_Prev_Switches : ARRAY[1..GVL_CONSTANTS.C_MAX_LIGHTING_ZONES] OF BOOL;
    L_Prev_Motion_Q : ARRAY[1..GVL_CONSTANTS.C_MAX_LIGHTING_ZONES] OF BOOL;
    L_Manual_Override : ARRAY[1..GVL_CONSTANTS.C_MAX_LIGHTING_ZONES] OF BOOL;
    L_Motion_Timers : ARRAY[1..GVL_CONSTANTS.C_MAX_LIGHTING_ZONES] OF FB_System_Timer_TOF;
    L_Rule_Light_Active : BOOL;
    L_Rule_Light_Val : BYTE;
    L_Rule_Blinds_Active : BOOL;
    L_Rule_Blinds_Val : BYTE;
    L_Wet_Zone_Idx : INT;
    L_Effective_Scenario : E_SCENARIO_TYPE;
    L_Effective_Simulation_Active : BOOL;
  END_VAR

      // Менеджер управления освещением и шторами/жалюзи.
// Обеспечивает работу по сценариями, датчикам движения, физическим выключателям и правилам.


IF NOT VI_IsActivePLC THEN RETURN; END_IF;

L_Lighting_V2_Shadow_Diff_Found := FALSE;
L_Blinds_V2_Shadow_Diff_Found := FALSE;
L_Blinds_V2_Switch_Enabled := TRUE;
L_Blinds_V2_Path_Ready := FALSE;
L_Blinds_Using_Legacy_Fallback := TRUE;
L_Lighting_V2_Switch_Enabled := TRUE;
L_Lighting_V2_Path_Ready := FALSE;
L_Lighting_Using_Legacy_Fallback := TRUE;

GVL_STATE.G_Lighting_IO_Fault := FALSE;
GVL_STATE.G_Lighting_Subsystem_Degraded := FALSE;

L_Effective_Scenario := VI_Current_Scenario;
L_Effective_Simulation_Active := VI_Simulation_Active;

CASE VI_System_Mode OF
    E_System_Operating_Mode.MODE_SAFE_STOP:
        FOR L_j := 1 TO GVL_CONSTANTS.C_MAX_LIGHTING_ZONES DO
            VO_Lighting_Levels[L_j] := 0;
        END_FOR;
        FOR L_j := 1 TO GVL_CONSTANTS.C_MAX_BLINDS DO
            VO_Blinds_Positions[L_j] := 100;
        END_FOR;
        FOR L_j := 1 TO GVL_CONSTANTS.C_MAX_WET_ZONES DO
            VO_Wet_Zone_Light_Active[L_j] := FALSE;
        END_FOR;
        RETURN;
    E_System_Operating_Mode.MODE_FREEZE_PROTECTION:
        L_Effective_Scenario := E_SCENARIO_TYPE.SCENARIO_NONE;
        L_Effective_Simulation_Active := FALSE;
    E_System_Operating_Mode.MODE_DEGRADED:
        L_Effective_Simulation_Active := FALSE;
END_CASE;

// Инициализация индекса мокрых зон
L_Wet_Zone_Idx := 1;
// Сброс массива мокрых зон
FOR L_i := 1 TO GVL_CONSTANTS.C_MAX_WET_ZONES DO
    VO_Wet_Zone_Light_Active[L_i] := FALSE;
END_FOR;

// Проверка связи с модулями ввода-вывода
FOR L_i := 1 TO GVL_CONSTANTS.C_MAX_MODULES DO
    IF NOT VI_IO_Modules_Online[L_i] THEN
        GVL_STATE.G_Lighting_IO_Fault := TRUE;
GVL_STATE.G_Lighting_Subsystem_Degraded := TRUE;
        // Переход в безопасное состояние при потере связи (свет выкл, шторы открыты для эвакуации)
        FOR L_j := 1 TO GVL_CONSTANTS.C_MAX_LIGHTING_ZONES DO
            VO_Lighting_Levels[L_j] := 0;
        END_FOR;
        FOR L_j := 1 TO GVL_CONSTANTS.C_MAX_BLINDS DO
            VO_Blinds_Positions[L_j] := 100;
        END_FOR;
        RETURN;
    END_IF;
END_FOR;

// 1. Определение целевых уровней по сценарию (ТЗ 7.1)
IF L_Effective_Scenario >= 1 AND L_Effective_Scenario <= GVL_CONSTANTS.C_MAX_SCENARIOS THEN
    L_Target_Base_Light := VI_Scenario_Configs[L_Effective_Scenario].lighting_level_base;
    L_Target_Base_Blinds := VI_Scenario_Configs[L_Effective_Scenario].blinds_position_percent;
ELSE
    L_Target_Base_Light := 100;
    L_Target_Base_Blinds := 100;
END_IF;

// Корректировка по астрономическому таймеру
IF VI_Is_Night AND L_Effective_Scenario <> E_SCENARIO_TYPE.SCENARIO_AWAY AND L_Effective_Scenario <> E_SCENARIO_TYPE.SCENARIO_SLEEP THEN
    L_Target_Base_Blinds := 0; // Закрывать шторы ночью
END_IF;

// Плавный переход при смене сценария
IF L_Effective_Scenario <> L_Prev_Scenario THEN
    L_Transition_Light(
        VI_System_Time := VI_System_Time_MS,
        VI_Start_Time := VI_System_Time_MS,
        VI_Duration := 5000, // 5 секунд на плавное изменение света
        VI_Start_Value := TO_REAL(L_Base_Light),
        VI_End_Value := TO_REAL(L_Target_Base_Light)
    );
    L_Transition_Blinds(
        VI_System_Time := VI_System_Time_MS,
        VI_Start_Time := VI_System_Time_MS,
        VI_Duration := 10000, // 10 секунд на плавное изменение штор
        VI_Start_Value := TO_REAL(L_Base_Blinds),
        VI_End_Value := TO_REAL(L_Target_Base_Blinds)
    );
    L_Prev_Scenario := L_Effective_Scenario;
ELSE
    L_Transition_Light(
        VI_System_Time := VI_System_Time_MS,
        VI_Start_Time := L_Transition_Light.VI_Start_Time,
        VI_Duration := L_Transition_Light.VI_Duration,
        VI_Start_Value := L_Transition_Light.VI_Start_Value,
        VI_End_Value := TO_REAL(L_Target_Base_Light)
    );
    L_Transition_Blinds(
        VI_System_Time := VI_System_Time_MS,
        VI_Start_Time := L_Transition_Blinds.VI_Start_Time,
        VI_Duration := L_Transition_Blinds.VI_Duration,
        VI_Start_Value := L_Transition_Blinds.VI_Start_Value,
        VI_End_Value := TO_REAL(L_Target_Base_Blinds)
    );
END_IF;

L_Base_Light := TO_BYTE(L_Transition_Light.VO_Current_Value);
L_Base_Blinds := TO_BYTE(L_Transition_Blinds.VO_Current_Value);

// 2. Управление освещением
FOR L_i := 1 TO GVL_CONSTANTS.C_MAX_LIGHTING_ZONES DO
    L_Rule_Light_Active := FALSE;
    L_Rule_Light_Val := 0;
    
    // Проверка правил
    FOR L_j := 1 TO GVL_CONSTANTS.C_MAX_RULES DO
        IF VI_Rule_Actions[L_j].Active AND VI_Rule_Actions[L_j].Target_ID = L_i THEN
            IF VI_Rule_Actions[L_j].Action_Type = E_Rule_Action_Type.ACTION_SET_LIGHTING_BASE THEN
                L_Rule_Light_Active := TRUE;
                L_Rule_Light_Val := REAL_TO_BYTE(VI_Rule_Actions[L_j].Value);
                L_Light_States[L_i] := (L_Rule_Light_Val > 0);
            ELSIF VI_Rule_Actions[L_j].Action_Type = E_Rule_Action_Type.ACTION_TOGGLE_LIGHTING AND VI_Rule_Actions[L_j].Triggered THEN
                L_Light_States[L_i] := NOT L_Light_States[L_i];
            END_IF;
        END_IF;
    END_FOR;

    // Приоритет 1: Физические выключатели (ТЗ 1.0)
    IF VI_Physical_Switches[L_i] AND NOT L_Prev_Switches[L_i] THEN
        L_Light_States[L_i] := NOT L_Light_States[L_i];
        L_Manual_Override[L_i] := TRUE; // Запоминаем ручное переопределение
    END_IF;
    L_Prev_Switches[L_i] := VI_Physical_Switches[L_i];

    // Приоритет 2: Датчики движения (ТЗ 2.0)
    // Защита от дребезга и удержание сигнала движения с помощью TOF
    L_Motion_Timers[L_i](IN := VI_Motion_Sensors[L_i], PT := T#5m, VI_System_Time_MS := VI_System_Time_MS);
    
    // Сброс ручного переопределения, когда комната становится пустой (задний фронт таймера движения)
    IF L_Prev_Motion_Q[L_i] AND NOT L_Motion_Timers[L_i].Q THEN
        L_Manual_Override[L_i] := FALSE;
    END_IF;
    L_Prev_Motion_Q[L_i] := L_Motion_Timers[L_i].Q;

    IF L_Motion_Timers[L_i].Q THEN
        IF NOT L_Manual_Override[L_i] THEN
            L_Light_States[L_i] := TRUE;
        END_IF;
    ELSE
        // Выключаем свет только если нет ручного переопределения
        IF NOT L_Manual_Override[L_i] THEN
            L_Light_States[L_i] := FALSE;
        END_IF;
    END_IF;

    // Приоритет 3: Симуляция (только в режиме Away)
    IF L_Effective_Scenario = E_SCENARIO_TYPE.SCENARIO_AWAY AND L_Effective_Simulation_Active THEN
        L_Light_States[L_i] := VI_Simulation_Lights[L_i];
    END_IF;

    // Приоритет 4: Ручное управление и правила
    IF VI_Manual_Light_Override[L_i] > 0 THEN
        VO_Lighting_Levels[L_i] := VI_Manual_Light_Override[L_i];
    ELSIF L_Rule_Light_Active THEN
        VO_Lighting_Levels[L_i] := L_Rule_Light_Val;
    ELSE
        VO_Lighting_Levels[L_i] := SEL(L_Light_States[L_i], 0, L_Base_Light);
    END_IF;
    
    // 5. Мокрые зоны
    IF VI_Wet_Zone_Map[L_i] AND L_Wet_Zone_Idx <= GVL_CONSTANTS.C_MAX_WET_ZONES THEN
        VO_Wet_Zone_Light_Active[L_Wet_Zone_Idx] := (VO_Lighting_Levels[L_i] > 10);
        L_Wet_Zone_Idx := L_Wet_Zone_Idx + 1;
    END_IF;
END_FOR;

// 3. Управление шторами
FOR L_i := 1 TO GVL_CONSTANTS.C_MAX_BLINDS DO
    L_Rule_Blinds_Active := FALSE;
    L_Rule_Blinds_Val := 0;
    
    // Проверка правил
    FOR L_j := 1 TO GVL_CONSTANTS.C_MAX_RULES DO
        IF VI_Rule_Actions[L_j].Active AND VI_Rule_Actions[L_j].Target_ID = L_i THEN
            IF VI_Rule_Actions[L_j].Action_Type = E_Rule_Action_Type.ACTION_SET_BLINDS THEN
                L_Rule_Blinds_Active := TRUE;
                L_Rule_Blinds_Val := REAL_TO_BYTE(VI_Rule_Actions[L_j].Value);
            END_IF;
        END_IF;
    END_FOR;

    // Приоритет 1: Ручное управление
    IF VI_Manual_Blinds_Override[L_i] > 0 THEN
        VO_Blinds_Positions[L_i] := VI_Manual_Blinds_Override[L_i];
    // Приоритет 2: Правила
    ELSIF L_Rule_Blinds_Active THEN
        VO_Blinds_Positions[L_i] := L_Rule_Blinds_Val;
    // Приоритет 3: Сценарий
    ELSE
        VO_Blinds_Positions[L_i] := L_Base_Blinds;
    END_IF;
END_FOR;

// ========================================
// Lighting V2 shadow execution (phase2)
// ========================================
fbLightingV2Staging(
    VI_Zone_ID := 1,
    VI_Enable := (VO_Lighting_Levels[1] > 0),
    VI_Brightness_Setpoint := BYTE_TO_REAL(VO_Lighting_Levels[1]),
    VI_Scene_ID := TO_INT(L_Effective_Scenario),
    VI_Manual_Override := (VI_Manual_Light_Override[1] > 0),
    VI_Transition_Time_MS := 5000,

    VI_Is_Active := (VO_Lighting_Levels[1] > 0),
    VI_Brightness_Actual := BYTE_TO_REAL(VO_Lighting_Levels[1]),
    VI_Motion_Active := VI_Motion_Sensors[1],
    VI_Ambient_Lux := 0.0,
    VI_Alarm_Active := GVL_STATE.G_Lighting_IO_Fault OR GVL_STATE.G_Lighting_Subsystem_Degraded,

    VO_Command_Shadow => L_Lighting_V2_Command_Shadow,
    VO_State_Shadow => L_Lighting_V2_State_Shadow
);

// ========================================
// Lighting V2 shadow validation
// ========================================
IF ABS(BYTE_TO_REAL(VO_Lighting_Levels[1]) - L_Lighting_V2_Command_Shadow.Brightness_Setpoint) > 0.1 THEN
    L_Lighting_V2_Shadow_Diff_Found := TRUE;
END_IF;
IF ABS(BYTE_TO_REAL(VO_Lighting_Levels[1]) - L_Lighting_V2_State_Shadow.Brightness_Actual) > 0.1 THEN
    L_Lighting_V2_Shadow_Diff_Found := TRUE;
END_IF;
IF VI_Motion_Sensors[1] <> L_Lighting_V2_State_Shadow.Motion_Active THEN
    L_Lighting_V2_Shadow_Diff_Found := TRUE;
END_IF;

// Guarded Lighting V2 enable
IF L_Lighting_V2_Switch_Enabled THEN
    IF NOT L_Lighting_V2_Shadow_Diff_Found THEN
        L_Lighting_V2_Path_Ready := TRUE;
        L_Lighting_Using_Legacy_Fallback := FALSE;
    ELSE
        L_Lighting_V2_Path_Ready := FALSE;
        L_Lighting_Using_Legacy_Fallback := TRUE;
    END_IF;
ELSE
    L_Lighting_V2_Path_Ready := FALSE;
    L_Lighting_Using_Legacy_Fallback := TRUE;
END_IF;



// ========================================
// Blinds V2 shadow execution (phase2)
// ========================================
fbBlindsV2Staging(
    VI_Blind_ID := 1,
    VI_Enable := TRUE,
    VI_Position_Setpoint := VO_Blinds_Positions[1],
    VI_Manual_Override := (VI_Manual_Blinds_Override[1] > 0),
    VI_Scenario_ID := TO_INT(L_Effective_Scenario),
    VI_Safety_Mode := FALSE,

    VI_Position_Actual := VO_Blinds_Positions[1],
    VI_Manual_Override_Active := (VI_Manual_Blinds_Override[1] > 0),
    VI_Is_Moving := FALSE,
    VI_Alarm_Active := GVL_STATE.G_Lighting_IO_Fault,

    VO_Command_Shadow => L_Blinds_V2_Command_Shadow,
    VO_State_Shadow => L_Blinds_V2_State_Shadow
);

// Blinds validation
IF VO_Blinds_Positions[1] <> L_Blinds_V2_Command_Shadow.Position_Setpoint THEN
    L_Blinds_V2_Shadow_Diff_Found := TRUE;
END_IF;
IF VO_Blinds_Positions[1] <> L_Blinds_V2_State_Shadow.Position_Actual THEN
    L_Blinds_V2_Shadow_Diff_Found := TRUE;
END_IF;


// Guarded Blinds V2 enable
IF L_Blinds_V2_Switch_Enabled THEN
    IF NOT L_Blinds_V2_Shadow_Diff_Found THEN
        L_Blinds_V2_Path_Ready := TRUE;
        L_Blinds_Using_Legacy_Fallback := FALSE;
    ELSE
        L_Blinds_V2_Path_Ready := FALSE;
        L_Blinds_Using_Legacy_Fallback := TRUE;
    END_IF;
ELSE
    L_Blinds_V2_Path_Ready := FALSE;
    L_Blinds_Using_Legacy_Fallback := TRUE;
END_IF;

// >>> BULK_SYNC_ANCHOR: FB_Lighting_Blinds_Manager <<<
    
END_FUNCTION_BLOCK

FUNCTION_BLOCK FB_NVRAM_Manager
  VAR_INPUT
    VI_Command : BYTE;
    VI_Offset : UDINT;
    VI_DataRef : REFERENCE TO BYTE;
    VI_DataSize : UDINT;
    VI_System_Time_MS : UDINT;
    VI_Operator_ID : STRING(10);
    VI_IsActivePLC : BOOL;
    VI_TwoPersonConfirmation : BOOL;
  END_VAR
  VAR_OUTPUT
    VO_Done : BOOL;
    VO_Error : BOOL;
    VO_ErrorID : UDINT;
    VO_ReadDataRef : REFERENCE TO BYTE;
    VO_HMI_Status_Message : STRING(200);
  END_VAR
  VAR
    L_prev_Command : BYTE;
    L_cmd_rising : BOOL;
    L_i : UDINT;
    L_Last_Write_Time_MS : UDINT := 0;
    L_Data_Changed : BOOL;
  END_VAR
  VAR
    C_MAX_NVRAM_SIZE : UDINT := 12800;
  END_VAR

      // Детекция фронта команды
L_cmd_rising := (VI_Command <> 0) AND (L_prev_Command = 0);
L_prev_Command := VI_Command;

IF L_cmd_rising THEN
    VO_Done := FALSE;
    VO_Error := FALSE;
    VO_ErrorID := 0;
    VO_HMI_Status_Message := '';
    
    // Валидация смещения
    IF VI_Offset >= C_MAX_NVRAM_SIZE THEN
        VO_Error := TRUE;
        VO_ErrorID := 16#1501;
        VO_HMI_Status_Message := 'NVRAM: Неверное смещение';
        VO_Done := TRUE;
        RETURN;
    END_IF;

    // Валидация указателя
    IF NOT __ISVALIDREF(VI_DataRef) THEN
        VO_Error := TRUE;
        VO_ErrorID := 16#150A;
        VO_HMI_Status_Message := 'NVRAM: Недействительная ссылка на данные';
        VO_Done := TRUE;
        RETURN;
    END_IF;

    IF (VI_Offset + VI_DataSize) > C_MAX_NVRAM_SIZE THEN
        VO_Error := TRUE;
        VO_ErrorID := 16#150B;
        VO_HMI_Status_Message := 'NVRAM: Размер данных превышает доступный объем';
        VO_Done := TRUE;
        RETURN;
    END_IF;

    IF VI_Command = 1 THEN // ЗАПИСЬ (WRITE)
        IF NOT VI_IsActivePLC THEN
            VO_Error := TRUE;
            VO_ErrorID := 16#1509;
            VO_HMI_Status_Message := 'NVRAM: Запись запрещена (STANDBY)';
        ELSE
            // Ограничение частоты записи (не чаще 1 раза в 60 секунд)
            IF F_TimeDiff(VI_System_Time_MS, L_Last_Write_Time_MS) < 60000 AND L_Last_Write_Time_MS <> 0 THEN
                VO_Error := TRUE;
                VO_ErrorID := 16#150C;
                VO_HMI_Status_Message := 'NVRAM: Превышена частота записи (лимит 1 раз в 60с)';
            ELSE
                // Проверка на изменение данных перед записью
                L_Data_Changed := FALSE;
                IF MEMCMP(ADR(GVL_Retain.G_NVRAM_Data[VI_Offset]), ADR(VI_DataRef), VI_DataSize) <> 0 THEN
                    L_Data_Changed := TRUE;
                END_IF;
                
                IF L_Data_Changed THEN
                    // Копируем данные используя MEMCPY
                    MEMCPY(ADR(GVL_Retain.G_NVRAM_Data[VI_Offset]), ADR(VI_DataRef), VI_DataSize);
                    L_Last_Write_Time_MS := VI_System_Time_MS;
                    VO_HMI_Status_Message := 'NVRAM: Данные успешно сохранены в RETAIN';
                ELSE
                    VO_HMI_Status_Message := 'NVRAM: Данные не изменились, запись пропущена';
                END_IF;
            END_IF;
        END_IF;
        VO_Done := TRUE;
        
    ELSIF VI_Command = 2 THEN // ЧТЕНИЕ (READ)
        // Копируем данные используя MEMCPY
        MEMCPY(ADR(VI_DataRef), ADR(GVL_Retain.G_NVRAM_Data[VI_Offset]), VI_DataSize);
        VO_ReadDataRef REF= VI_DataRef;
        VO_HMI_Status_Message := 'NVRAM: Данные успешно прочитаны из RETAIN';
        VO_Done := TRUE;
    END_IF;
END_IF;

IF VI_Command = 0 THEN
    VO_Done := FALSE;
END_IF;
// >>> BULK_SYNC_ANCHOR: FB_NVRAM_Manager <<<
    
END_FUNCTION_BLOCK

FUNCTION_BLOCK FB_PID_Controller
  VAR_INPUT
    VI_SetPoint : REAL;
    VI_ProcessValue : REAL;
    VI_Kp : REAL;
    VI_Tn : REAL;
    VI_Tv : REAL;
    VI_Y_Min : REAL := 0.0;
    VI_Y_Max : REAL := 100.0;
    VI_Manual_Mode : BOOL;
    VI_Manual_Value : REAL;
    VI_Deadband : REAL := 0.1;
    VI_Cycle_Time_S : REAL := 0.01;
    VI_Reset : BOOL;
  END_VAR
  VAR_OUTPUT
    VO_Output : REAL;
    VO_Error : REAL;
    VO_Limiting : BOOL;
  END_VAR
  VAR
    L_Integral_Sum : REAL;
    L_Prev_Error : REAL;
    L_Derivative : REAL;
    L_Output_Raw : REAL;
  END_VAR

      // Расчет ошибки
VO_Error := VI_SetPoint - VI_ProcessValue;

// Проверка мертвой зоны
IF ABS(VO_Error) < VI_Deadband THEN
    VO_Error := 0.0;
END_IF;

IF VI_Reset THEN
    L_Integral_Sum := 0.0;
    L_Prev_Error := 0.0;
    VO_Output := 0.0;
    RETURN;
END_IF;

IF VI_Manual_Mode THEN
    VO_Output := VI_Manual_Value;
    // Безударный переход: при выходе из ручного режима выход должен остаться прежним.
    // Так как Выход = P + I + D, то I = Выход - P - D.
    // Для простоты D при переходе обнуляем (или игнорируем), тогда I = Выход - P.
    L_Integral_Sum := VO_Output - (VI_Kp * VO_Error);
    L_Prev_Error := VO_Error;
    RETURN;
END_IF;

// Пропорциональная составляющая
L_Output_Raw := VI_Kp * VO_Error;

// Интегральная составляющая (Метод трапеций)
IF VI_Tn > 0.0 THEN
    // Anti-windup: не накапливаем интеграл, если выход уже на пределе и ошибка того же знака
    IF NOT VO_Limiting OR (VO_Error > 0.0 AND L_Output_Raw < VI_Y_Max) OR (VO_Error < 0.0 AND L_Output_Raw > VI_Y_Min) THEN
        L_Integral_Sum := L_Integral_Sum + (VI_Kp / VI_Tn) * VO_Error * VI_Cycle_Time_S;
    END_IF;
    L_Output_Raw := L_Output_Raw + L_Integral_Sum;
END_IF;

// Дифференциальная составляющая
IF VI_Tv > 0.0 THEN
    L_Derivative := (VO_Error - L_Prev_Error) / VI_Cycle_Time_S;
    L_Output_Raw := L_Output_Raw + VI_Kp * VI_Tv * L_Derivative;
END_IF;

L_Prev_Error := VO_Error;

// Ограничение выхода
IF L_Output_Raw > VI_Y_Max THEN
    VO_Output := VI_Y_Max;
    VO_Limiting := TRUE;
ELSIF L_Output_Raw < VI_Y_Min THEN
    VO_Output := VI_Y_Min;
    VO_Limiting := TRUE;
ELSE
    VO_Output := L_Output_Raw;
    VO_Limiting := FALSE;
END_IF;
// >>> BULK_SYNC_ANCHOR: FB_PID_Controller <<<
    
END_FUNCTION_BLOCK

FUNCTION_BLOCK FB_Redundancy_Manager
  VAR_INPUT
    VI_System_Time_MS : UDINT;
    VI_Local_PLC_ID : BYTE;
    VI_Remote_Pulse : BOOL;
    VI_Remote_Is_Active : BOOL;
    VI_Gateway_Ping_OK : BOOL;
    VI_Remote_State : ST_System_State_Snapshot;
    VI_Local_State : ST_System_State_Snapshot;
  END_VAR
  VAR_OUTPUT
    VO_Local_Role : E_PLC_ROLE;
    VO_Local_Pulse : BOOL;
    VO_Sync_Data_Req : BOOL;
    VO_Status_Msg : STRING(200);
    VO_Synced_State : ST_System_State_Snapshot;
    VO_State_Updated : BOOL;
  END_VAR
  VAR
    L_Heartbeat : FB_PLC_Heartbeat;
    L_Pulse_Timer : FB_System_Timer;
    L_Pulse_State : BOOL;
    L_Prev_Role : E_PLC_ROLE;
    L_State_Replicator : FB_State_Replication;
  END_VAR

      // 1. Генерация собственного пульса (меандр 100 мс)
L_Pulse_Timer(IN := NOT L_Pulse_Timer.Q, PT := T#100ms, VI_System_Time_MS := VI_System_Time_MS);
IF L_Pulse_Timer.Q THEN
    L_Pulse_State := NOT L_Pulse_State;
END_IF;
VO_Local_Pulse := L_Pulse_State;

// 2. Определение роли через Heartbeat
L_Heartbeat(
    VI_Local_ID := VI_Local_PLC_ID,
    VI_System_Time := VI_System_Time_MS,
    VI_Remote_Pulse := VI_Remote_Pulse,
    VI_Remote_Is_Active := VI_Remote_Is_Active,
    VI_Gateway_Ping_OK := VI_Gateway_Ping_OK
);

IF L_Heartbeat.VO_Is_Active THEN
    VO_Local_Role := E_PLC_ROLE.ROLE_ACTIVE;
    VO_Status_Msg := 'ПЛК АКТИВЕН (ВЕДУЩИЙ)';
ELSE
    VO_Local_Role := E_PLC_ROLE.ROLE_STANDBY;
    VO_Status_Msg := 'ПЛК В РЕЗЕРВЕ (ВЕДОМЫЙ)';
END_IF;

// 3. Запрос на синхронизацию при переходе в ACTIVE
IF VO_Local_Role = E_PLC_ROLE.ROLE_ACTIVE AND L_Prev_Role = E_PLC_ROLE.ROLE_STANDBY THEN
    VO_Sync_Data_Req := TRUE;
ELSE
    VO_Sync_Data_Req := FALSE;
END_IF;

L_State_Replicator(
    VI_Local_Role := VO_Local_Role,
    VI_Sync_Req := VO_Sync_Data_Req,
    VI_Local_State := VI_Local_State,
    VI_Remote_State := VI_Remote_State,
    VI_System_Time_MS := VI_System_Time_MS
);
VO_Synced_State := L_State_Replicator.VO_Synced_State;
VO_State_Updated := L_State_Replicator.VO_State_Updated;

L_Prev_Role := VO_Local_Role;
// >>> BULK_SYNC_ANCHOR: FB_Redundancy_Manager <<<
    
END_FUNCTION_BLOCK

FUNCTION_BLOCK FB_Rule_Engine
  VAR_INPUT
    VI_System_Time_MS : UDINT;
    VI_IsActivePLC : BOOL;
    VI_Security_Armed : BOOL;
    VI_Current_Time : TOD;
    VI_Day_Of_Week : INT;
  END_VAR
  VAR_OUTPUT
    VO_Actions : ARRAY[1..GVL_CONSTANTS.C_MAX_RULES] OF ST_Rule_Action;
  END_VAR
  VAR_IN_OUT
    VI_Rules : ARRAY[1..GVL_CONSTANTS.C_MAX_RULES] OF ST_User_Rule;
    VI_Indoor_Temps : ARRAY[1..GVL_CONSTANTS.C_MAX_CLIMATE_ZONES] OF REAL;
    VI_Floor_Temps : ARRAY[1..GVL_CONSTANTS.C_MAX_HEATING_CIRCUITS] OF REAL;
    VI_Humidities : ARRAY[1..GVL_CONSTANTS.C_MAX_CLIMATE_ZONES] OF REAL;
    VI_CO2_Levels : ARRAY[1..GVL_CONSTANTS.C_MAX_CLIMATE_ZONES] OF REAL;
    VI_Motion_Sensors : ARRAY[1..GVL_CONSTANTS.C_MAX_CLIMATE_ZONES] OF BOOL;
    VI_Door_Sensors : ARRAY[1..GVL_CONSTANTS.C_MAX_DOOR_SENSORS] OF BOOL;
    VI_Window_Sensors : ARRAY[1..GVL_CONSTANTS.C_MAX_CLIMATE_ZONES] OF BOOL;
    VI_Water_Sensors : ARRAY[1..GVL_CONSTANTS.C_MAX_FLOOD_SENSORS] OF BOOL;
    VI_Smoke_Sensors : ARRAY[1..GVL_CONSTANTS.C_MAX_SMOKE_SENSORS] OF BOOL;
    VI_Methane_Sensors : ARRAY[1..GVL_CONSTANTS.C_MAX_METHANE_SENSORS] OF REAL;
    VI_CO_Sensors : ARRAY[1..GVL_CONSTANTS.C_MAX_CO_SENSORS] OF REAL;
  END_VAR
  VAR
    L_i : INT;
    fbCompat : ARRAY[1..GVL_CONSTANTS.C_MAX_RULES] OF FB_Rule_Compatibility_Package;
    L_Compat_All_OK : BOOL;
    L_Compat_First_Warning : STRING(255);
    L_Compat_First_Warning_Latched : BOOL;
    L_Shadow_V2_Enabled : BOOL;
    L_Shadow_V2_Roundtrip_Mismatch : BOOL;
    L_Shadow_V2_First_Mismatch_Rule : INT;
    L_V2_Switch_Enabled : BOOL;
    L_V2_Path_Ready : BOOL;
    L_V2_Using_Legacy_Fallback : BOOL;
    L_Condition_Met : BOOL;
    L_Current_Value : REAL;
    L_Triggers : ARRAY[1..GVL_CONSTANTS.C_MAX_RULES] OF R_TRIG;
    L_Trigger_Count : ARRAY[1..GVL_CONSTANTS.C_MAX_RULES] OF UINT;
    L_Last_Reset_Time : UDINT;
    L_Elapsed_Time : UDINT;
  END_VAR

      IF NOT VI_IsActivePLC THEN RETURN; END_IF;

L_Compat_All_OK := TRUE;
L_Compat_First_Warning := '';
L_Compat_First_Warning_Latched := FALSE;
L_Shadow_V2_Enabled := TRUE;
L_Shadow_V2_Roundtrip_Mismatch := FALSE;
L_Shadow_V2_First_Mismatch_Rule := 0;
L_V2_Switch_Enabled := FALSE;
L_V2_Path_Ready := FALSE;
L_V2_Using_Legacy_Fallback := TRUE;

// Сброс счетчиков срабатываний каждую минуту (защита от циклических зависимостей/дребезга)
L_Elapsed_Time := F_TimeDiff(VI_System_Time_MS, L_Last_Reset_Time);

IF L_Elapsed_Time >= GVL_CONSTANTS.C_MS_IN_MINUTE THEN
    L_Last_Reset_Time := VI_System_Time_MS;
    FOR L_i := 1 TO GVL_CONSTANTS.C_MAX_RULES DO
        L_Trigger_Count[L_i] := 0;
    END_FOR;
END_IF;

FOR L_i := 1 TO GVL_CONSTANTS.C_MAX_RULES DO
    fbCompat[L_i](VI_Rule_Legacy := VI_Rules[L_i]);

    IF NOT fbCompat[L_i].VO_Forward_OK OR NOT fbCompat[L_i].VO_Reverse_OK THEN
        L_Compat_All_OK := FALSE;
    END_IF;

    IF (NOT L_Compat_First_Warning_Latched) AND (fbCompat[L_i].VO_Warning_Text <> '') THEN
        L_Compat_First_Warning := fbCompat[L_i].VO_Warning_Text;
        L_Compat_First_Warning_Latched := TRUE;
    END_IF;

    IF L_Shadow_V2_Enabled THEN
        IF (fbCompat[L_i].VO_Rule_Legacy_Roundtrip.Action_Type <> VI_Rules[L_i].Action_Type)
           OR (fbCompat[L_i].VO_Rule_Legacy_Roundtrip.Action_Target_ID <> VI_Rules[L_i].Action_Target_ID)
           OR (ABS(fbCompat[L_i].VO_Rule_Legacy_Roundtrip.Action_Value - VI_Rules[L_i].Action_Value) > 0.0001)
           OR (fbCompat[L_i].VO_Rule_Legacy_Roundtrip.Condition_Type <> VI_Rules[L_i].Condition_Type)
           OR (fbCompat[L_i].VO_Rule_Legacy_Roundtrip.Condition_Target_ID <> VI_Rules[L_i].Condition_Target_ID)
           OR (fbCompat[L_i].VO_Rule_Legacy_Roundtrip.Condition_Op <> VI_Rules[L_i].Condition_Op)
           OR (ABS(fbCompat[L_i].VO_Rule_Legacy_Roundtrip.Condition_Value - VI_Rules[L_i].Condition_Value) > 0.0001)
           OR (ABS(fbCompat[L_i].VO_Rule_Legacy_Roundtrip.Condition_Value_Max - VI_Rules[L_i].Condition_Value_Max) > 0.0001) THEN
            L_Shadow_V2_Roundtrip_Mismatch := TRUE;
            IF L_Shadow_V2_First_Mismatch_Rule = 0 THEN
                L_Shadow_V2_First_Mismatch_Rule := L_i;
            END_IF;
        END_IF;
    END_IF;

    // Phase 4 scaffold: optional V2 switch point.
    // Current state: always remain on legacy behavior.
    // Future state: when V2 path is implemented and validated,
    // this block becomes the controlled branch point.
    IF L_V2_Switch_Enabled AND L_V2_Path_Ready THEN
        L_V2_Using_Legacy_Fallback := FALSE;
        // V2 action-generation path placeholder.
        // No runtime behavior change yet.
    ELSE
        L_V2_Using_Legacy_Fallback := TRUE;
    END_IF;

    VO_Actions[L_i].Active := FALSE;
    IF VI_Rules[L_i].Enabled THEN
        L_Condition_Met := FALSE;
        L_Current_Value := 0.0;
        
        // Определение значения для проверки
        IF VI_Rules[L_i].Condition_Target_ID > 0 THEN
            CASE VI_Rules[L_i].Condition_Type OF
                E_Rule_Condition_Type.COND_AIR_TEMP: IF VI_Rules[L_i].Condition_Target_ID <= GVL_CONSTANTS.C_MAX_CLIMATE_ZONES THEN L_Current_Value := VI_Indoor_Temps[VI_Rules[L_i].Condition_Target_ID]; END_IF;
                E_Rule_Condition_Type.COND_FLOOR_TEMP: IF VI_Rules[L_i].Condition_Target_ID <= GVL_CONSTANTS.C_MAX_HEATING_CIRCUITS THEN L_Current_Value := VI_Floor_Temps[VI_Rules[L_i].Condition_Target_ID]; END_IF;
                E_Rule_Condition_Type.COND_HUMIDITY: IF VI_Rules[L_i].Condition_Target_ID <= GVL_CONSTANTS.C_MAX_CLIMATE_ZONES THEN L_Current_Value := VI_Humidities[VI_Rules[L_i].Condition_Target_ID]; END_IF;
                E_Rule_Condition_Type.COND_CO2: IF VI_Rules[L_i].Condition_Target_ID <= GVL_CONSTANTS.C_MAX_CLIMATE_ZONES THEN L_Current_Value := VI_CO2_Levels[VI_Rules[L_i].Condition_Target_ID]; END_IF;
                E_Rule_Condition_Type.COND_MOTION: IF VI_Rules[L_i].Condition_Target_ID <= GVL_CONSTANTS.C_MAX_CLIMATE_ZONES THEN L_Current_Value := SEL(VI_Motion_Sensors[VI_Rules[L_i].Condition_Target_ID], 0.0, 1.0); END_IF;
                E_Rule_Condition_Type.COND_DOOR_WINDOW: 
                    IF VI_Rules[L_i].Condition_Target_ID <= GVL_CONSTANTS.C_MAX_DOOR_SENSORS THEN
                        L_Current_Value := SEL(VI_Door_Sensors[VI_Rules[L_i].Condition_Target_ID] OR VI_Window_Sensors[VI_Rules[L_i].Condition_Target_ID], 0.0, 1.0);
                    ELSIF VI_Rules[L_i].Condition_Target_ID <= GVL_CONSTANTS.C_MAX_CLIMATE_ZONES THEN
                        L_Current_Value := SEL(VI_Window_Sensors[VI_Rules[L_i].Condition_Target_ID], 0.0, 1.0);
                    END_IF;
                E_Rule_Condition_Type.COND_FLOOD: IF VI_Rules[L_i].Condition_Target_ID <= GVL_CONSTANTS.C_MAX_FLOOD_SENSORS THEN L_Current_Value := SEL(VI_Water_Sensors[VI_Rules[L_i].Condition_Target_ID], 0.0, 1.0); END_IF;
                E_Rule_Condition_Type.COND_SMOKE: IF VI_Rules[L_i].Condition_Target_ID <= GVL_CONSTANTS.C_MAX_SMOKE_SENSORS THEN L_Current_Value := SEL(VI_Smoke_Sensors[VI_Rules[L_i].Condition_Target_ID], 0.0, 1.0); END_IF;
                E_Rule_Condition_Type.COND_METHANE: IF VI_Rules[L_i].Condition_Target_ID <= GVL_CONSTANTS.C_MAX_METHANE_SENSORS THEN L_Current_Value := VI_Methane_Sensors[VI_Rules[L_i].Condition_Target_ID]; END_IF;
                E_Rule_Condition_Type.COND_CO: IF VI_Rules[L_i].Condition_Target_ID <= GVL_CONSTANTS.C_MAX_CO_SENSORS THEN L_Current_Value := VI_CO_Sensors[VI_Rules[L_i].Condition_Target_ID]; END_IF;
                E_Rule_Condition_Type.COND_TIME_OF_DAY: L_Current_Value := TO_REAL(TOD_TO_UDINT(VI_Current_Time) / GVL_CONSTANTS.C_MS_IN_MINUTE); // Время в минутах
                E_Rule_Condition_Type.COND_DAY_OF_WEEK: L_Current_Value := TO_REAL(VI_Day_Of_Week);
            END_CASE;
        ELSE
            IF VI_Rules[L_i].Condition_Type = E_Rule_Condition_Type.COND_TIME_OF_DAY THEN
                L_Current_Value := TO_REAL(TOD_TO_UDINT(VI_Current_Time) / GVL_CONSTANTS.C_MS_IN_MINUTE); // Время в минутах
            ELSIF VI_Rules[L_i].Condition_Type = E_Rule_Condition_Type.COND_DAY_OF_WEEK THEN
                L_Current_Value := TO_REAL(VI_Day_Of_Week);
            END_IF;
        END_IF;
        
        // Проверка условия
        CASE VI_Rules[L_i].Condition_Op OF
            E_Rule_Comparison.COMP_GT: L_Condition_Met := (L_Current_Value > VI_Rules[L_i].Condition_Value);
            E_Rule_Comparison.COMP_LT: L_Condition_Met := (L_Current_Value < VI_Rules[L_i].Condition_Value);
            E_Rule_Comparison.COMP_EQ: L_Condition_Met := (ABS(L_Current_Value - VI_Rules[L_i].Condition_Value) < 0.1);
            E_Rule_Comparison.COMP_GE: L_Condition_Met := (L_Current_Value >= VI_Rules[L_i].Condition_Value);
            E_Rule_Comparison.COMP_LE: L_Condition_Met := (L_Current_Value <= VI_Rules[L_i].Condition_Value);
            E_Rule_Comparison.COMP_IN_RANGE: L_Condition_Met := (L_Current_Value >= VI_Rules[L_i].Condition_Value) AND (L_Current_Value <= VI_Rules[L_i].Condition_Value_Max);
            E_Rule_Comparison.COMP_TRUE: L_Condition_Met := (L_Current_Value > 0.5);
            E_Rule_Comparison.COMP_FALSE: L_Condition_Met := (L_Current_Value < 0.5);
        END_CASE;
        
        // Формирование действия
        L_Triggers[L_i](CLK := L_Condition_Met);
        
        IF L_Triggers[L_i].Q THEN
            L_Trigger_Count[L_i] := L_Trigger_Count[L_i] + 1;
            IF L_Trigger_Count[L_i] > 10 THEN
                // ТЗ 13.5: Блокировка правила при слишком частом срабатывании (циклическая зависимость)
                VO_Actions[L_i].Active := FALSE;
                VO_Actions[L_i].Triggered := FALSE;
                CONTINUE; // Пропускаем выполнение
            END_IF;
        END_IF;
        
        IF L_Condition_Met AND (L_Trigger_Count[L_i] <= 10) THEN
            VO_Actions[L_i].Active := TRUE;
            VO_Actions[L_i].Triggered := L_Triggers[L_i].Q;
            VO_Actions[L_i].Action_Type := VI_Rules[L_i].Action_Type;
            VO_Actions[L_i].Target_ID := VI_Rules[L_i].Action_Target_ID;
            VO_Actions[L_i].Value := VI_Rules[L_i].Action_Value;
        END_IF;
    END_IF;
END_FOR;
// >>> BULK_SYNC_ANCHOR: FB_Rule_Engine <<<
    
END_FUNCTION_BLOCK

FUNCTION_BLOCK FB_Safety_Manager
  VAR_INPUT
    VI_Gas_Alarm : BOOL;
    VI_Leak_Alarm : BOOL;
    VI_Smoke_Alarm : BOOL;
    VI_Reset : BOOL;
  END_VAR
  VAR_OUTPUT
    VO_Gas_Latched : BOOL;
    VO_Leak_Latched : BOOL;
    VO_Smoke_Latched : BOOL;
    VO_Emergency_Stop : BOOL;
  END_VAR
  VAR
    L_Any_Active : BOOL;
  END_VAR

      // Защёлкиваем аварии независимо друг от друга
IF VI_Gas_Alarm THEN
    VO_Gas_Latched := TRUE;
END_IF;

IF VI_Leak_Alarm THEN
    VO_Leak_Latched := TRUE;
END_IF;

IF VI_Smoke_Alarm THEN
    VO_Smoke_Latched := TRUE;
END_IF;

L_Any_Active := VI_Gas_Alarm OR VI_Leak_Alarm OR VI_Smoke_Alarm;

// Ручной сброс допустим только когда все входные аварийные сигналы уже исчезли
IF VI_Reset AND NOT L_Any_Active THEN
    VO_Gas_Latched := FALSE;
    VO_Leak_Latched := FALSE;
    VO_Smoke_Latched := FALSE;
END_IF;

// Агрегированный аварийный стоп = любая защёлкнутая safety-авария
VO_Emergency_Stop := VO_Gas_Latched OR VO_Leak_Latched OR VO_Smoke_Latched;

// >>> BULK_SYNC_ANCHOR: FB_Safety_Manager <<<
    
END_FUNCTION_BLOCK

FUNCTION_BLOCK FB_Scenario_Manager
  VAR_INPUT
    VI_System_Time_MS : UDINT;
    VI_Activate_Request : E_SCENARIO_TYPE;
    VI_IsActivePLC : BOOL;
    VI_System_Mode : E_System_Operating_Mode;
  END_VAR
  VAR_OUTPUT
    VO_Current_Scenario : E_SCENARIO_TYPE;
    VO_Status_Msg : STRING(200);
  END_VAR
  VAR
    L_Last_Scenario_Time : UDINT;
  END_VAR

      IF NOT VI_IsActivePLC THEN
    RETURN;
END_IF;

CASE VI_System_Mode OF
    E_System_Operating_Mode.MODE_SAFE_STOP,
    E_System_Operating_Mode.MODE_FREEZE_PROTECTION:
        IF VO_Current_Scenario <> E_SCENARIO_TYPE.SCENARIO_NONE THEN
            VO_Current_Scenario := E_SCENARIO_TYPE.SCENARIO_NONE;
            VO_Status_Msg := 'Сценарии принудительно отключены режимом безопасности';
        END_IF;
        RETURN;

    E_System_Operating_Mode.MODE_DEGRADED:
        VO_Status_Msg := 'Смена сценариев заблокирована: деградированный режим';
        RETURN;
END_CASE;

IF VI_Activate_Request <> VO_Current_Scenario THEN
    // Проверка минимального времени работы сценария
    IF F_TimeDiff(VI_System_Time_MS, L_Last_Scenario_Time) >= 60000 OR VO_Current_Scenario = E_SCENARIO_TYPE.SCENARIO_NONE THEN
        // Логика переключения сценариев
        VO_Current_Scenario := VI_Activate_Request;
        L_Last_Scenario_Time := VI_System_Time_MS;
        
        CASE VO_Current_Scenario OF
        E_SCENARIO_TYPE.SCENARIO_NONE:
            VO_Status_Msg := 'Сценарии отключены';
        E_SCENARIO_TYPE.SCENARIO_AWAY:
            VO_Status_Msg := 'Активирован сценарий: Вне дома (Охрана + Энергосбережение)';
        E_SCENARIO_TYPE.SCENARIO_SLEEP:
            VO_Status_Msg := 'Активирован сценарий: Сон (Ночное освещение + Климат)';
        E_SCENARIO_TYPE.SCENARIO_PRESENCE:
            VO_Status_Msg := 'Активирован сценарий: Имитация присутствия';
        END_CASE;
    END_IF;
END_IF;
// >>> BULK_SYNC_ANCHOR: FB_Scenario_Manager <<<
    
END_FUNCTION_BLOCK

FUNCTION_BLOCK FB_Security_System_Manager
  VAR_INPUT
    VI_System_Time_MS : UDINT;
    VI_IsActivePLC : BOOL;
    VI_Arm_Request : BOOL;
    VI_Disarm_Request : BOOL;
    VI_PIN_Code : STRING(4);
    VI_RFID_Tag : STRING(20);
    VI_2FA_Code : STRING(6);
    VI_Config : ST_Security_Global_Config;
    VI_Current_TOD : TOD;
  END_VAR
  VAR_OUTPUT
    VO_Armed : BOOL;
    VO_Alarm_Active : BOOL;
    VO_Siren_Active : BOOL;
    VO_Status_Msg : STRING(200);
    VO_Send_Code_Req : BOOL;
    VO_Code_To_Send : STRING(6);
  END_VAR
  VAR_IN_OUT
    VI_Motion_Sensors : ARRAY[1..GVL_CONSTANTS.C_MAX_CLIMATE_ZONES] OF BOOL;
    VI_Door_Sensors : ARRAY[1..GVL_CONSTANTS.C_MAX_DOOR_SENSORS] OF BOOL;
    VI_Window_Sensors : ARRAY[1..GVL_CONSTANTS.C_MAX_CLIMATE_ZONES] OF BOOL;
    VI_Bypass_Motion : ARRAY[1..GVL_CONSTANTS.C_MAX_CLIMATE_ZONES] OF BOOL;
    VI_Bypass_Doors : ARRAY[1..GVL_CONSTANTS.C_MAX_DOOR_SENSORS] OF BOOL;
    VI_Bypass_Windows : ARRAY[1..GVL_CONSTANTS.C_MAX_CLIMATE_ZONES] OF BOOL;
  END_VAR
  VAR
    L_i : INT;
    L_Any_Sensor_Active : BOOL;
    L_Arm_Delay_Timer : FB_System_Timer;
    L_Alarm_Delay_Timer : FB_System_Timer;
    L_Arming_In_Progress : BOOL;
    L_Valid_PIN : BOOL;
    fbAccessCode : FB_AccessCode_Manager;
    fbTwoFactor : FB_TwoFactor_Auth;
    L_2FA_Required : BOOL;
    L_Disarm_Pending : BOOL;
    L_Reset_2FA : BOOL;
    L_Auto_Arm_Trigger : BOOL;
    R_Trig_Auto_Arm : R_TRIG;
  END_VAR

      IF NOT VI_IsActivePLC THEN RETURN; END_IF;

// 1. Проверка PIN-кода или RFID-метки через менеджер кодов
fbAccessCode(
    VI_System_Time_MS := VI_System_Time_MS,
    VI_IsActivePLC := VI_IsActivePLC,
    VI_Code_To_Check := VI_PIN_Code,
    VI_RFID_To_Check := VI_RFID_Tag,
    VO_Code_Valid => L_Valid_PIN
);

// 2. Логика постановки на охрану (с задержкой на выход)
L_Auto_Arm_Trigger := FALSE;
IF VI_Config.auto_arm_enabled THEN
    IF VI_Current_TOD >= UDINT_TO_TOD(VI_Config.auto_arm_time_ms) THEN
        L_Auto_Arm_Trigger := TRUE;
    END_IF;
END_IF;
R_Trig_Auto_Arm(CLK := L_Auto_Arm_Trigger);

IF ((VI_Arm_Request AND L_Valid_PIN) OR R_Trig_Auto_Arm.Q) AND NOT VO_Armed AND NOT L_Arming_In_Progress THEN
    // Проверка, что все двери/окна закрыты перед постановкой (с учетом байпаса)
    L_Any_Sensor_Active := FALSE;
    FOR L_i := 1 TO GVL_CONSTANTS.C_MAX_DOOR_SENSORS DO IF VI_Door_Sensors[L_i] AND NOT VI_Bypass_Doors[L_i] THEN L_Any_Sensor_Active := TRUE; END_IF; END_FOR;
    FOR L_i := 1 TO GVL_CONSTANTS.C_MAX_CLIMATE_ZONES DO IF VI_Window_Sensors[L_i] AND NOT VI_Bypass_Windows[L_i] THEN L_Any_Sensor_Active := TRUE; END_IF; END_FOR;
    
    IF NOT L_Any_Sensor_Active THEN
        L_Arming_In_Progress := TRUE;
        VO_Status_Msg := 'Постановка на охрану. Покиньте помещение.';
    ELSE
        VO_Status_Msg := 'Ошибка постановки: Открыты двери или окна';
    END_IF;
END_IF;

L_Arm_Delay_Timer(IN := L_Arming_In_Progress, PT := TO_TIME(VI_Config.exit_delay_seconds * 1000), VI_System_Time_MS := VI_System_Time_MS);
IF L_Arm_Delay_Timer.Q THEN
    L_Arming_In_Progress := FALSE;
    VO_Armed := TRUE;
    VO_Status_Msg := 'Система под охраной';
END_IF;

// 3. Логика снятия с охраны с 2FA
IF VI_Disarm_Request AND L_Valid_PIN AND VO_Armed THEN
    IF VI_Config.enable_2fa THEN
        L_Disarm_Pending := TRUE;
        L_2FA_Required := TRUE;
        VO_Status_Msg := 'Ожидание 2FA для снятия с охраны';
    ELSE
        // Снятие без 2FA
        VO_Armed := FALSE;
        VO_Alarm_Active := FALSE;
        VO_Siren_Active := FALSE;
        L_Arming_In_Progress := FALSE;
        VO_Status_Msg := 'Система снята с охраны';
    END_IF;
END_IF;

fbTwoFactor(
    VI_System_Time_MS := VI_System_Time_MS,
    VI_Start_Auth := L_2FA_Required,
    VI_Method := E_TwoFactor_Method.TF_METHOD_TOTP, // Для примера
    VI_User_Code := VI_2FA_Code, // Используем отдельный вход для 2FA кода
    VI_Reset_Success := L_Reset_2FA
);

VO_Send_Code_Req := fbTwoFactor.VO_Send_Code_Req;
VO_Code_To_Send := fbTwoFactor.VO_Code_To_Send;

IF L_Disarm_Pending AND fbTwoFactor.VO_State.Is_Success THEN
    VO_Armed := FALSE;
    VO_Alarm_Active := FALSE;
    VO_Siren_Active := FALSE;
    L_Arming_In_Progress := FALSE;
    L_Disarm_Pending := FALSE;
    L_2FA_Required := FALSE;
    L_Reset_2FA := TRUE;
    VO_Status_Msg := 'Система снята с охраны';
ELSIF L_Disarm_Pending AND fbTwoFactor.VO_State.Is_Locked THEN
    L_Disarm_Pending := FALSE;
    L_2FA_Required := FALSE;
    L_Reset_2FA := FALSE;
    VO_Status_Msg := 'Ошибка 2FA: Превышено количество попыток';
ELSE
    L_Reset_2FA := FALSE;
END_IF;

// 4. Логика тревоги (с задержкой на вход)
IF VO_Armed THEN
    L_Any_Sensor_Active := FALSE;
    FOR L_i := 1 TO GVL_CONSTANTS.C_MAX_CLIMATE_ZONES DO IF VI_Motion_Sensors[L_i] AND NOT VI_Bypass_Motion[L_i] THEN L_Any_Sensor_Active := TRUE; END_IF; END_FOR;
    FOR L_i := 1 TO GVL_CONSTANTS.C_MAX_DOOR_SENSORS DO IF VI_Door_Sensors[L_i] AND NOT VI_Bypass_Doors[L_i] THEN L_Any_Sensor_Active := TRUE; END_IF; END_FOR;
    FOR L_i := 1 TO GVL_CONSTANTS.C_MAX_CLIMATE_ZONES DO IF VI_Window_Sensors[L_i] AND NOT VI_Bypass_Windows[L_i] THEN L_Any_Sensor_Active := TRUE; END_IF; END_FOR;
    
    // Защелкиваем факт нарушения периметра, чтобы кратковременное срабатывание датчика не сбрасывало таймер
    IF L_Any_Sensor_Active THEN
        L_Alarm_Delay_Timer.IN := TRUE;
    END_IF;
    
    L_Alarm_Delay_Timer(PT := TO_TIME(VI_Config.entry_delay_seconds * 1000), VI_System_Time_MS := VI_System_Time_MS);
    
    IF L_Alarm_Delay_Timer.Q THEN
        VO_Alarm_Active := TRUE;
        VO_Siren_Active := TRUE;
        VO_Status_Msg := 'ТРЕВОГА! Нарушение периметра';
    ELSIF L_Alarm_Delay_Timer.IN THEN
        VO_Status_Msg := 'Внимание! Введите PIN-код для отмены тревоги';
    END_IF;
ELSE
    L_Alarm_Delay_Timer(IN := FALSE, PT := T#0s, VI_System_Time_MS := VI_System_Time_MS); // Сброс таймера при снятии с охраны
END_IF;
// >>> BULK_SYNC_ANCHOR: FB_Security_System_Manager <<<
    
END_FUNCTION_BLOCK

FUNCTION_BLOCK FB_Simulation_Manager
  VAR_INPUT
    VI_System_Time_MS : UDINT;
    VI_IsActivePLC : BOOL;
    VI_Scenario : E_SCENARIO_TYPE;
    VI_Config : ST_Scenario_Config;
  END_VAR
  VAR_OUTPUT
    VO_Sim_Lights : ARRAY[1..GVL_CONSTANTS.C_MAX_LIGHTING_ZONES] OF BOOL;
    VO_Sim_Active : BOOL;
    VO_Sim_Water_Leak : ARRAY[1..GVL_CONSTANTS.C_MAX_FLOOD_SENSORS] OF BOOL;
    VO_Sim_Gas_Leak : ARRAY[1..GVL_CONSTANTS.C_MAX_METHANE_SENSORS] OF REAL;
  END_VAR
  VAR
    L_Random : FB_Random_Generator;
    L_Last_Toggle : UDINT;
    L_i : INT;
    L_Rand_Val : UDINT;
    L_Test_Mode : BOOL := FALSE;
  END_VAR

      IF VI_Scenario = E_SCENARIO_TYPE.SCENARIO_AWAY AND VI_Config.Presence_Simulation_Enabled THEN
    VO_Sim_Active := TRUE;
    
    // Переключаем свет каждые 30 минут
    IF F_TimeDiff(VI_System_Time_MS, L_Last_Toggle) >= (GVL_CONSTANTS.C_MS_IN_MINUTE * 30) THEN
        L_Last_Toggle := VI_System_Time_MS;
        
        FOR L_i := 1 TO GVL_CONSTANTS.C_MAX_LIGHTING_ZONES DO
            L_Rand_Val := L_Random.Random_Int_Range(VI_min := 0, VI_max := 100);
            VO_Sim_Lights[L_i] := (L_Rand_Val > 80); // 20% шанс включения
        END_FOR;
    END_IF;
ELSE
    VO_Sim_Active := FALSE;
    FOR L_i := 1 TO GVL_CONSTANTS.C_MAX_LIGHTING_ZONES DO VO_Sim_Lights[L_i] := FALSE; END_FOR;
END_IF;

// Симуляция аварий в тестовом режиме
IF L_Test_Mode THEN
    // Генерация случайных протечек (очень редко)
    L_Rand_Val := L_Random.Random_Int_Range(VI_min := 0, VI_max := 100000);
    IF L_Rand_Val = 42 THEN
        VO_Sim_Water_Leak[1] := TRUE;
    END_IF;
    
    // Симуляция утечки газа
    L_Rand_Val := L_Random.Random_Int_Range(VI_min := 0, VI_max := 100000);
    IF L_Rand_Val = 77 THEN
        VO_Sim_Gas_Leak[1] := 15.0; // 15% LEL
    END_IF;
ELSE
    FOR L_i := 1 TO GVL_CONSTANTS.C_MAX_FLOOD_SENSORS DO VO_Sim_Water_Leak[L_i] := FALSE; END_FOR;
    FOR L_i := 1 TO GVL_CONSTANTS.C_MAX_METHANE_SENSORS DO VO_Sim_Gas_Leak[L_i] := 0.0; END_FOR;
END_IF;
// >>> BULK_SYNC_ANCHOR: FB_Simulation_Manager <<<
    
END_FUNCTION_BLOCK

FUNCTION_BLOCK FB_Socket_Manager
  VAR_INPUT
    VI_System_Time_MS : UDINT;
    VI_IsActivePLC : BOOL;
    VI_Scenario : E_SCENARIO_TYPE;
    VI_Fire_Alarm : BOOL;
    VI_Flood_Alarm : BOOL;
    VI_Security_Armed : BOOL;
  END_VAR
  VAR_OUTPUT
    VO_Socket_States : ARRAY[1..GVL_CONSTANTS.C_MAX_SOCKETS] OF BOOL;
    VO_Internal_States : ARRAY[1..GVL_CONSTANTS.C_MAX_SOCKETS] OF BOOL;
  END_VAR
  VAR_IN_OUT
    VI_Manual_Override : ARRAY[1..GVL_CONSTANTS.C_MAX_SOCKETS] OF BOOL;
    VI_Physical_Switches : ARRAY[1..GVL_CONSTANTS.C_MAX_SOCKETS] OF BOOL;
    VI_Rule_Actions : ARRAY[1..GVL_CONSTANTS.C_MAX_RULES] OF ST_Rule_Action;
    VI_IO_Modules_Online : ARRAY[1..GVL_CONSTANTS.C_MAX_MODULES] OF BOOL;
  END_VAR
  VAR
    fbSocketV2Staging : FB_Socket_V2_Staging;
    L_Socket_V2_Command_Shadow : ST_Socket_Command_V2;
    L_Socket_V2_State_Shadow : ST_Socket_State_V2;
    L_Socket_V2_Shadow_Diff_Found : BOOL;
    L_Socket_V2_Switch_Enabled : BOOL;
    L_Socket_V2_Path_Ready : BOOL;
    L_Socket_Using_Legacy_Fallback : BOOL;
    L_i : INT;
    L_j : INT;
    L_Rule_State : BOOL;
    L_Rule_Active : BOOL;
    L_Internal_State : ARRAY[1..GVL_CONSTANTS.C_MAX_SOCKETS] OF BOOL;
    L_Manual_Trig : ARRAY[1..GVL_CONSTANTS.C_MAX_SOCKETS] OF R_TRIG;
  END_VAR

      // Менеджер управления розетками.
// Обеспечивает работу по сценариям, правилам и аварийное отключение (без локальных выключателей розеток).


IF NOT VI_IsActivePLC THEN RETURN; END_IF;

L_Socket_V2_Shadow_Diff_Found := FALSE;
L_Socket_V2_Switch_Enabled := TRUE;
L_Socket_V2_Path_Ready := FALSE;
L_Socket_Using_Legacy_Fallback := TRUE;

// Проверка связи с модулями ввода-вывода
FOR L_i := 1 TO GVL_CONSTANTS.C_MAX_MODULES DO
    IF NOT VI_IO_Modules_Online[L_i] THEN
        // Переход в безопасное состояние при потере связи (отключение всех розеток)
        FOR L_j := 1 TO GVL_CONSTANTS.C_MAX_SOCKETS DO
            VO_Socket_States[L_j] := FALSE;
        END_FOR;
        RETURN;
    END_IF;
END_FOR;

FOR L_i := 1 TO GVL_CONSTANTS.C_MAX_SOCKETS DO
    L_Rule_Active := FALSE;
    L_Rule_State := FALSE;
    
    L_Manual_Trig[L_i](CLK := VI_Manual_Override[L_i]);
    
    // Ручное переключение
    IF L_Manual_Trig[L_i].Q THEN
        L_Internal_State[L_i] := NOT L_Internal_State[L_i];
    END_IF;

    // Проверка правил для текущей розетки
    FOR L_j := 1 TO GVL_CONSTANTS.C_MAX_RULES DO
        IF VI_Rule_Actions[L_j].Active AND VI_Rule_Actions[L_j].Target_ID = L_i THEN
            IF VI_Rule_Actions[L_j].Action_Type = E_Rule_Action_Type.ACTION_SET_SOCKET THEN
                L_Rule_Active := TRUE;
                L_Rule_State := (VI_Rule_Actions[L_j].Value > 0.5);
                L_Internal_State[L_i] := L_Rule_State; // Синхронизация внутреннего состояния
            ELSIF VI_Rule_Actions[L_j].Action_Type = E_Rule_Action_Type.ACTION_TOGGLE_SOCKET AND VI_Rule_Actions[L_j].Triggered THEN
                L_Internal_State[L_i] := NOT L_Internal_State[L_i]; // Toggle
            END_IF;
        END_IF;
    END_FOR;

    // Аварийное отключение
    IF VI_Fire_Alarm OR VI_Flood_Alarm THEN
        // Розетки 1-4 неотключаемые (холодильник, сервер и т.д.)
        IF L_i > 4 THEN
            VO_Socket_States[L_i] := FALSE;
        ELSE
            // Критические розетки сохраняют свое текущее внутреннее состояние, а не форсируются в TRUE
            VO_Socket_States[L_i] := L_Internal_State[L_i];
        END_IF;
    ELSIF VI_Scenario = E_SCENARIO_TYPE.SCENARIO_AWAY OR VI_Security_Armed THEN
        // Master Off
        IF L_i > 4 THEN
            VO_Socket_States[L_i] := FALSE;
        ELSE
            // Неотключаемые розетки могут управляться вручную
            VO_Socket_States[L_i] := L_Internal_State[L_i];
        END_IF;
    ELSE
        // Нормальный режим: состояние определяется внутренним состоянием (ручным или правилом)
        IF L_Rule_Active THEN
            VO_Socket_States[L_i] := L_Rule_State;
        ELSE
            VO_Socket_States[L_i] := L_Internal_State[L_i];
        END_IF;
    END_IF;
END_FOR;

VO_Internal_States := L_Internal_State;

// ========================================
// Socket V2 shadow execution (phase2)
// ========================================
fbSocketV2Staging(
    VI_Socket_ID := 1,
    VI_Enable := TRUE,
    VI_Target_State := VO_Socket_States[1],
    VI_Manual_Override := VI_Manual_Override[1],
    VI_Safety_Lock := (VI_Fire_Alarm OR VI_Flood_Alarm),
    VI_Scenario_ID := TO_INT(VI_Scenario),

    VI_Is_On := VO_Socket_States[1],
    VI_Manual_Override_Active := VI_Manual_Override[1],
    VI_Safety_Blocked := (VI_Fire_Alarm OR VI_Flood_Alarm),
    VI_Alarm_Active := (VI_Fire_Alarm OR VI_Flood_Alarm),

    VO_Command_Shadow => L_Socket_V2_Command_Shadow,
    VO_State_Shadow => L_Socket_V2_State_Shadow
);

// ========================================
// Socket V2 shadow validation
// ========================================
IF VO_Socket_States[1] <> L_Socket_V2_Command_Shadow.Target_State THEN
    L_Socket_V2_Shadow_Diff_Found := TRUE;
END_IF;
IF VO_Socket_States[1] <> L_Socket_V2_State_Shadow.Is_On THEN
    L_Socket_V2_Shadow_Diff_Found := TRUE;
END_IF;
IF (VI_Fire_Alarm OR VI_Flood_Alarm) <> L_Socket_V2_State_Shadow.Safety_Blocked THEN
    L_Socket_V2_Shadow_Diff_Found := TRUE;
END_IF;

// Guarded Socket V2 enable
IF L_Socket_V2_Switch_Enabled THEN
    IF NOT L_Socket_V2_Shadow_Diff_Found THEN
        L_Socket_V2_Path_Ready := TRUE;
        L_Socket_Using_Legacy_Fallback := FALSE;
    ELSE
        L_Socket_V2_Path_Ready := FALSE;
        L_Socket_Using_Legacy_Fallback := TRUE;
    END_IF;
ELSE
    L_Socket_V2_Path_Ready := FALSE;
    L_Socket_Using_Legacy_Fallback := TRUE;
END_IF;

// >>> BULK_SYNC_ANCHOR: FB_Socket_Manager <<<
    
END_FUNCTION_BLOCK

FUNCTION_BLOCK FB_State_Manager
  VAR_INPUT
    VI_System_Severity : E_System_Severity;
    VI_Root_Cause : E_System_Root_Cause;
    VI_Freeze_Risk : BOOL := FALSE;
  END_VAR
  VAR_OUTPUT
    VO_System_OK : BOOL;
    VO_System_Warning : BOOL;
    VO_System_Critical : BOOL;
    VO_Status_Msg : STRING(200);
    VO_System_Mode : E_System_Operating_Mode;
  END_VAR

      VO_System_OK := FALSE;
VO_System_Warning := FALSE;
VO_System_Critical := FALSE;
VO_Status_Msg := '';
VO_System_Mode := E_System_Operating_Mode.MODE_NORMAL;

CASE VI_System_Severity OF
    E_System_Severity.SEV_NORMAL:
        VO_System_OK := TRUE;
        VO_Status_Msg := 'Система в норме';
        VO_System_Mode := E_System_Operating_Mode.MODE_NORMAL;

    E_System_Severity.SEV_WARNING:
        VO_System_Warning := TRUE;
        VO_System_Mode := E_System_Operating_Mode.MODE_DEGRADED;
        CASE VI_Root_Cause OF
            E_System_Root_Cause.ROOT_WATER_LEAK:
                VO_Status_Msg := 'Предупреждение: протечка воды';
            E_System_Root_Cause.ROOT_CO_WARNING:
                VO_Status_Msg := 'Предупреждение: повышенный CO';
            ELSE
                VO_Status_Msg := 'Предупреждение системы';
        END_CASE;

    E_System_Severity.SEV_DEGRADED:
        VO_System_Warning := TRUE;
        VO_System_Mode := E_System_Operating_Mode.MODE_DEGRADED;
        CASE VI_Root_Cause OF
            E_System_Root_Cause.ROOT_SENSOR_FAULT:
                VO_Status_Msg := 'Деградация: ошибка датчика';
            E_System_Root_Cause.ROOT_IO_OFFLINE:
                VO_Status_Msg := 'Деградация: модуль IO недоступен';
            E_System_Root_Cause.ROOT_COMM_FAULT:
                VO_Status_Msg := 'Деградация: ошибка связи';
            E_System_Root_Cause.ROOT_WATCHDOG_FAULT:
                VO_Status_Msg := 'Деградация: watchdog fault';
            E_System_Root_Cause.ROOT_SUBSYSTEM_FAULT:
                VO_Status_Msg := 'Деградация: ошибка подсистемы';
            ELSE
                VO_Status_Msg := 'Деградация системы';
        END_CASE;

    E_System_Severity.SEV_CRITICAL:
        VO_System_Critical := TRUE;

        IF (VI_Root_Cause = E_System_Root_Cause.ROOT_GAS_LEAK OR
            VI_Root_Cause = E_System_Root_Cause.ROOT_CO_CRITICAL) AND
            VI_Freeze_Risk THEN
            VO_System_Mode := E_System_Operating_Mode.MODE_FREEZE_PROTECTION;
        ELSE
            VO_System_Mode := E_System_Operating_Mode.MODE_SAFE_STOP;
        END_IF;

        CASE VI_Root_Cause OF
            E_System_Root_Cause.ROOT_FIRE:
                VO_Status_Msg := 'АВАРИЯ: ПОЖАР';
            E_System_Root_Cause.ROOT_GAS_LEAK:
                VO_Status_Msg := 'АВАРИЯ: УТЕЧКА ГАЗА';
            E_System_Root_Cause.ROOT_CO_CRITICAL:
                VO_Status_Msg := 'АВАРИЯ: КРИТИЧЕСКИЙ CO';
            E_System_Root_Cause.ROOT_WATCHDOG_FAULT:
                VO_Status_Msg := 'АВАРИЯ: WATCHDOG';
            ELSE
                VO_Status_Msg := 'АВАРИЯ СИСТЕМЫ';
        END_CASE;
END_CASE;
// >>> BULK_SYNC_ANCHOR: FB_State_Manager <<<
    
END_FUNCTION_BLOCK

FUNCTION_BLOCK FB_System_Health
  VAR_INPUT
    VI_Smoke_Detected : BOOL;
    VI_Gas_Detected : BOOL;
    VI_CO_Warning_Level : BOOL;
    VI_CO_Alarm_Level : BOOL;
    VI_Leak_Detected : BOOL;
    VI_Sensor_Fault : BOOL := FALSE;
    VI_IO_Offline : BOOL := FALSE;
    VI_Comm_Fault : BOOL := FALSE;
    VI_Watchdog_Fault : BOOL := FALSE;
    VI_Subsystem_Fault : BOOL := FALSE;
  END_VAR
  VAR_OUTPUT
    VO_System_Severity : E_System_Severity;
    VO_Root_Cause : E_System_Root_Cause;
    VO_Sensor_Fault : BOOL;
    VO_IO_Fault : BOOL;
    VO_Comm_Fault : BOOL;
    VO_Subsystem_Degraded : BOOL;
    VO_First_Fault_Active : BOOL;
    VO_First_Fault_Type : INT;
    VO_First_Fault_Source : INT;
  END_VAR

      VO_Sensor_Fault := VI_Sensor_Fault;
VO_IO_Fault := VI_IO_Offline;
VO_Comm_Fault := VI_Comm_Fault;
VO_Subsystem_Degraded := VI_Subsystem_Fault;

VO_System_Severity := E_System_Severity.SEV_NORMAL;
VO_Root_Cause := E_System_Root_Cause.ROOT_NONE;
VO_First_Fault_Active := FALSE;
VO_First_Fault_Type := 0;
VO_First_Fault_Source := 0;

// Priority: FIRE > GAS > CO > WATER > diagnostics
IF VI_Smoke_Detected THEN
    VO_System_Severity := E_System_Severity.SEV_CRITICAL;
    VO_Root_Cause := E_System_Root_Cause.ROOT_FIRE;
    VO_First_Fault_Active := TRUE;
    VO_First_Fault_Type := 5;

ELSIF VI_Gas_Detected THEN
    VO_System_Severity := E_System_Severity.SEV_CRITICAL;
    VO_Root_Cause := E_System_Root_Cause.ROOT_GAS_LEAK;
    VO_First_Fault_Active := TRUE;
    VO_First_Fault_Type := 6;

ELSIF VI_CO_Alarm_Level THEN
    VO_System_Severity := E_System_Severity.SEV_CRITICAL;
    VO_Root_Cause := E_System_Root_Cause.ROOT_CO_CRITICAL;
    VO_First_Fault_Active := TRUE;
    VO_First_Fault_Type := 7;

ELSIF VI_CO_Warning_Level THEN
    VO_System_Severity := E_System_Severity.SEV_WARNING;
    VO_Root_Cause := E_System_Root_Cause.ROOT_CO_WARNING;
    VO_First_Fault_Active := TRUE;
    VO_First_Fault_Type := 7;

ELSIF VI_Leak_Detected THEN
    VO_System_Severity := E_System_Severity.SEV_WARNING;
    VO_Root_Cause := E_System_Root_Cause.ROOT_WATER_LEAK;
    VO_First_Fault_Active := TRUE;
    VO_First_Fault_Type := 8;

ELSIF VI_Watchdog_Fault THEN
    VO_System_Severity := E_System_Severity.SEV_CRITICAL;
    VO_Root_Cause := E_System_Root_Cause.ROOT_WATCHDOG_FAULT;
    VO_First_Fault_Active := TRUE;
    VO_First_Fault_Type := 9;

ELSIF VI_IO_Offline THEN
    VO_System_Severity := E_System_Severity.SEV_DEGRADED;
    VO_Root_Cause := E_System_Root_Cause.ROOT_IO_OFFLINE;
    VO_First_Fault_Active := TRUE;
    VO_First_Fault_Type := 1;

ELSIF VI_Comm_Fault THEN
    VO_System_Severity := E_System_Severity.SEV_DEGRADED;
    VO_Root_Cause := E_System_Root_Cause.ROOT_COMM_FAULT;
    VO_First_Fault_Active := TRUE;
    VO_First_Fault_Type := 3;

ELSIF VI_Sensor_Fault THEN
    VO_System_Severity := E_System_Severity.SEV_DEGRADED;
    VO_Root_Cause := E_System_Root_Cause.ROOT_SENSOR_FAULT;
    VO_First_Fault_Active := TRUE;
    VO_First_Fault_Type := 2;

ELSIF VI_Subsystem_Fault THEN
    VO_System_Severity := E_System_Severity.SEV_DEGRADED;
    VO_Root_Cause := E_System_Root_Cause.ROOT_SUBSYSTEM_FAULT;
    VO_First_Fault_Active := TRUE;
    VO_First_Fault_Type := 4;
END_IF;
// >>> BULK_SYNC_ANCHOR: FB_System_Health <<<
    
END_FUNCTION_BLOCK

FUNCTION_BLOCK FB_System_Timer
  VAR_INPUT
    IN : BOOL;
    PT : TIME;
    VI_System_Time_MS : UDINT;
  END_VAR
  VAR_OUTPUT
    Q : BOOL;
    ET : TIME;
  END_VAR
  VAR
    L_Start_Time : UDINT;
    L_Running : BOOL;
  END_VAR

      // ==============================================================================
// Блок таймера, привязанный к системному времени (System Timer)
// Назначение:
// - Замена стандартного TON для обеспечения точной выдержки времени,
//   независимой от времени цикла ПЛК, с использованием единого системного времени.
// ==============================================================================



IF IN THEN
    IF NOT L_Running THEN
        L_Start_Time := VI_System_Time_MS;
        L_Running := TRUE;
        ET := T#0s;
        Q := FALSE;
    ELSE
        // Обработка переполнения UDINT (примерно 49 дней)
        ET := TO_TIME(F_TimeDiff(VI_System_Time_MS, L_Start_Time));
        
        IF ET >= PT THEN
            Q := TRUE;
            ET := PT;
        ELSE
            Q := FALSE;
        END_IF;
    END_IF;
ELSE
    L_Running := FALSE;
    ET := T#0s;
    Q := FALSE;
END_IF;
// >>> BULK_SYNC_ANCHOR: FB_System_Timer <<<
    
END_FUNCTION_BLOCK

FUNCTION_BLOCK FB_Ventilation_System_Manager
  VAR_INPUT
    VI_System_Time_MS : UDINT;
    VI_IsActivePLC : BOOL;
    VI_Outdoor_Temp : REAL;
    VI_Current_Scenario : E_SCENARIO_TYPE;
    VI_System_Mode : E_System_Operating_Mode;
    VI_Config : ST_Ventilation_Global_Config;
    VI_Fire_Alarm : BOOL;
    VI_Gas_Alarm : BOOL;
    VI_PV3_Boost_Req : BOOL;
    VI_Supply_100_Req : BOOL;
    VI_Exhaust_100_Req : BOOL;
    VI_Supply_80_Req : BOOL;
    VI_Vent_Stop : BOOL;
    VI_IO_Modules_Online : ARRAY[1..GVL_CONSTANTS.C_MAX_MODULES] OF BOOL;
  END_VAR
  VAR_OUTPUT
    VO_Supply_Fans : ARRAY[1..GVL_CONSTANTS.C_MAX_SUPPLY_FANS] OF BYTE;
    VO_Exhaust_Fans : ARRAY[1..GVL_CONSTANTS.C_MAX_EXHAUST_FANS] OF BYTE;
    VO_Heater_Power : ARRAY[1..GVL_CONSTANTS.C_MAX_BOILERS] OF REAL;
    VO_Status_Msg : STRING(200);
  END_VAR
  VAR_IN_OUT
    VI_Supply_Temps : ARRAY[1..GVL_CONSTANTS.C_MAX_SUPPLY_TEMPS] OF REAL;
    VI_Room_Temps : ARRAY[1..GVL_CONSTANTS.C_MAX_CLIMATE_ZONES] OF REAL;
    VI_Room_Humidities : ARRAY[1..GVL_CONSTANTS.C_MAX_CLIMATE_ZONES] OF REAL;
    VI_Room_CO2 : ARRAY[1..GVL_CONSTANTS.C_MAX_CLIMATE_ZONES] OF REAL;
    VI_Wet_Zone_Active : ARRAY[1..GVL_CONSTANTS.C_MAX_WET_ZONES] OF BOOL;
    VI_Rule_Actions : ARRAY[1..GVL_CONSTANTS.C_MAX_RULES] OF ST_Rule_Action;
  END_VAR
  VAR
    L_Policy_Normal : BOOL;
    L_Policy_Safe_Stop : BOOL;
    L_Policy_Degraded : BOOL;
    L_Policy_Freeze_Protection : BOOL;
    L_i : INT;
    L_j : INT;
    L_Max_CO2 : REAL;
    L_Max_Hum : REAL;
    L_Base_Speed : BYTE;
    L_Target_Temp : REAL;
    L_PID_Heaters : ARRAY[1..GVL_CONSTANTS.C_MAX_BOILERS] OF FB_PID_Controller;
    L_Wet_Zone_Timers : ARRAY[1..GVL_CONSTANTS.C_MAX_WET_ZONES] OF FB_System_Timer_TOF;
    fbVentilationV2Staging : FB_Ventilation_V2_Staging;
    L_Vent_Command_Shadow : ST_Ventilation_Command_V2;
    L_Vent_State_Shadow : ST_Ventilation_State_V2;
    L_Vent_V2_Shadow_Diff_Found : BOOL;
    L_Vent_V2_Switch_Enabled : BOOL;
    L_Vent_V2_Path_Ready : BOOL;
    L_Vent_Using_Legacy_Fallback : BOOL;
  END_VAR

      // ========================================
// Ventilation policy layer (phase3/v2)
// ========================================
GVL_STATE.G_Ventilation_IO_Fault := FALSE;
GVL_STATE.G_Ventilation_Subsystem_Degraded := FALSE;
L_Vent_V2_Shadow_Diff_Found := FALSE;
L_Vent_V2_Switch_Enabled := TRUE;
L_Vent_V2_Path_Ready := FALSE;
L_Vent_Using_Legacy_Fallback := TRUE;
L_Policy_Normal := (VI_System_Mode = E_System_Operating_Mode.MODE_NORMAL);
L_Policy_Safe_Stop := (VI_System_Mode = E_System_Operating_Mode.MODE_SAFE_STOP);
L_Policy_Degraded := (VI_System_Mode = E_System_Operating_Mode.MODE_DEGRADED);
L_Policy_Freeze_Protection := (VI_System_Mode = E_System_Operating_Mode.MODE_FREEZE_PROTECTION);

IF NOT VI_IsActivePLC THEN
    FOR L_i := 1 TO GVL_CONSTANTS.C_MAX_SUPPLY_FANS DO
        VO_Supply_Fans[L_i] := 0;
        IF L_i <= GVL_CONSTANTS.C_MAX_SUPPLY_TEMPS THEN
            VO_Heater_Power[L_i] := 0.0;
        END_IF;
    END_FOR;
    FOR L_i := 1 TO GVL_CONSTANTS.C_MAX_EXHAUST_FANS DO
        VO_Exhaust_Fans[L_i] := 0;
    END_FOR;
    VO_Status_Msg := 'ВЕНТИЛЯЦИЯ: РЕЗЕРВНЫЙ ПЛК';
    RETURN;
END_IF;

// Проверка связи с модулями ввода-вывода
FOR L_i := 1 TO GVL_CONSTANTS.C_MAX_MODULES DO
    IF NOT VI_IO_Modules_Online[L_i] THEN
        GVL_STATE.G_Ventilation_IO_Fault := TRUE;
        // Переход в безопасное состояние при потере связи (отключение вентиляции)
        FOR L_j := 1 TO GVL_CONSTANTS.C_MAX_SUPPLY_FANS DO
            VO_Supply_Fans[L_j] := 0;
        END_FOR;
        FOR L_j := 1 TO GVL_CONSTANTS.C_MAX_EXHAUST_FANS DO
            VO_Exhaust_Fans[L_j] := 0;
        END_FOR;
        FOR L_j := 1 TO GVL_CONSTANTS.C_MAX_BOILERS DO
            VO_Heater_Power[L_j] := 0.0;
        END_FOR;
        VO_Status_Msg := 'ОШИБКА: Потеря связи с модулями ввода-вывода';
        RETURN;
    END_IF;
END_FOR;

// =========================
// SYSTEM MODE OVERRIDE
// =========================
// VENT_POLICY_ROUTING_PHASE3_V2
IF L_Policy_Safe_Stop THEN
    FOR L_i := 1 TO GVL_CONSTANTS.C_MAX_SUPPLY_FANS DO
        VO_Supply_Fans[L_i] := 0;
    END_FOR;
    FOR L_i := 1 TO GVL_CONSTANTS.C_MAX_EXHAUST_FANS DO
        VO_Exhaust_Fans[L_i] := 0;
    END_FOR;
    FOR L_i := 1 TO GVL_CONSTANTS.C_MAX_BOILERS DO
        VO_Heater_Power[L_i] := 0.0;
    END_FOR;
    VO_Status_Msg := 'ВЕНТИЛЯЦИЯ: ОСТАНОВЛЕНА POLICY SAFE_STOP';
    RETURN;
END_IF;

IF L_Policy_Degraded THEN
    FOR L_i := 1 TO GVL_CONSTANTS.C_MAX_SUPPLY_FANS DO
        VO_Supply_Fans[L_i] := 0;
    END_FOR;
    FOR L_i := 1 TO GVL_CONSTANTS.C_MAX_BOILERS DO
        VO_Heater_Power[L_i] := 0.0;
    END_FOR;
    GVL_STATE.G_Ventilation_Subsystem_Degraded := TRUE;
    VO_Status_Msg := 'ВЕНТИЛЯЦИЯ: DEGRADED POLICY';
END_IF;

IF L_Policy_Freeze_Protection THEN
    FOR L_i := 1 TO GVL_CONSTANTS.C_MAX_SUPPLY_FANS DO
        VO_Supply_Fans[L_i] := 0;
    END_FOR;
    FOR L_i := 1 TO GVL_CONSTANTS.C_MAX_EXHAUST_FANS DO
        VO_Exhaust_Fans[L_i] := 0;
    END_FOR;
    FOR L_i := 1 TO GVL_CONSTANTS.C_MAX_BOILERS DO
        VO_Heater_Power[L_i] := 0.0;
    END_FOR;
    VO_Status_Msg := 'ВЕНТИЛЯЦИЯ: FREEZE_PROTECTION POLICY (stop)';
    RETURN;
END_IF;

// MODE_FREEZE_PROTECTION пока оставляем на текущей штатной логике

// 1. Определение базовой скорости и целевой температуры по сценарию (ТЗ 7.1)
CASE VI_Current_Scenario OF
    E_SCENARIO_TYPE.SCENARIO_AWAY:
        L_Base_Speed := VI_Config.Scenario_Modes[3].Base_Fan_Speed;
        L_Target_Temp := VI_Config.Scenario_Modes[3].Target_Temp;
    E_SCENARIO_TYPE.SCENARIO_SLEEP:
        L_Base_Speed := VI_Config.Scenario_Modes[2].Base_Fan_Speed;
        L_Target_Temp := VI_Config.Scenario_Modes[2].Target_Temp;
    ELSE // PRESENCE, MORNING, EVENING
        L_Base_Speed := VI_Config.Scenario_Modes[1].Base_Fan_Speed;
        L_Target_Temp := VI_Config.Scenario_Modes[1].Target_Temp;
END_CASE;

// 2. Логика управления приточными установками (П-1, П-2, П-3)
FOR L_i := 1 TO GVL_CONSTANTS.C_MAX_SUPPLY_FANS DO
    // ПИД-регулирование мощности электрического калорифера
    IF L_i <= GVL_CONSTANTS.C_MAX_SUPPLY_TEMPS THEN
        L_PID_Heaters[L_i](
            VI_SetPoint := L_Target_Temp,
            VI_ProcessValue := VI_Supply_Temps[L_i], // Используем датчик температуры после калорифера
            VI_Kp := 4.0, VI_Tn := 120.0, VI_Tv := 0.0,
            VI_Y_Min := 0.0, VI_Y_Max := 100.0, VI_Cycle_Time_S := 1.0,
            VO_Output => VO_Heater_Power[L_i]
        );
    END_IF;

    // Определение скорости приточного вентилятора
    VO_Supply_Fans[L_i] := L_Base_Speed;
    
    // Обработка действий от Rule Engine
    FOR L_j := 1 TO GVL_CONSTANTS.C_MAX_RULES DO
        IF VI_Rule_Actions[L_j].Active AND VI_Rule_Actions[L_j].Target_ID = L_i THEN
            IF VI_Rule_Actions[L_j].Action_Type = E_Rule_Action_Type.ACTION_SET_VENTILATION THEN
                VO_Supply_Fans[L_i] := REAL_TO_BYTE(VI_Rule_Actions[L_j].Value);
            END_IF;
        END_IF;
    END_FOR;
    
    // Requests are observed but must not bypass policy directly.
    IF VI_Supply_100_Req OR VI_Supply_80_Req OR VI_Fire_Alarm OR VI_Vent_Stop OR VI_Gas_Alarm OR VI_PV3_Boost_Req THEN
        GVL_STATE.G_Ventilation_Subsystem_Degraded := TRUE;
    END_IF;
END_FOR;

// 3. Логика управления вытяжными установками (В-1 .. В-5)
FOR L_i := 1 TO GVL_CONSTANTS.C_MAX_EXHAUST_FANS DO
    VO_Exhaust_Fans[L_i] := L_Base_Speed;
    
    // ТЗ 4.0: Логика вытяжки в санузлах
    FOR L_j := 1 TO GVL_CONSTANTS.C_MAX_WET_ZONES DO
        IF VI_Config.wet_zone_to_exhaust_map[L_j] = L_i THEN
            // Включение по свету, выключение с задержкой 5 минут (используем TOF)
            L_Wet_Zone_Timers[L_j](IN := VI_Wet_Zone_Active[L_j], PT := T#5m, VI_System_Time_MS := VI_System_Time_MS);
            IF VI_Wet_Zone_Active[L_j] THEN
                VO_Exhaust_Fans[L_i] := 80; // Повышенная скорость при присутствии
            ELSIF L_Wet_Zone_Timers[L_j].Q THEN
                VO_Exhaust_Fans[L_i] := 50; // Скорость выбега (пока таймер TOF активен)
            END_IF;
        END_IF;
    END_FOR;

    // Requests are observed but must not bypass policy directly.
    IF (L_i = VI_Config.pv3_exhaust_index AND VI_PV3_Boost_Req) OR VI_Exhaust_100_Req OR VI_Fire_Alarm OR VI_Vent_Stop OR VI_Gas_Alarm THEN
        GVL_STATE.G_Ventilation_Subsystem_Degraded := TRUE;
    END_IF;
END_FOR;








// ========================================
// VENT_FINAL_CLAMP
// ========================================
IF L_Policy_Degraded THEN
    FOR L_i := 1 TO GVL_CONSTANTS.C_MAX_EXHAUST_FANS DO
        VO_Exhaust_Fans[L_i] := MIN(VO_Exhaust_Fans[L_i], VI_Config.Degraded_Exhaust_Limit);
    END_FOR;
END_IF;

// Ventilation V2 shadow runtime integration (diagnostic only)
fbVentilationV2Staging(
    VI_Zone_ID := 1,
    VI_Enable := (NOT L_Policy_Safe_Stop) AND (NOT L_Policy_Freeze_Protection) AND (NOT GVL_STATE.G_Ventilation_IO_Fault),
    VI_Fan_Speed_Setpoint := BYTE_TO_REAL(VO_Supply_Fans[1]),
    VI_Damper_Position_Setpoint := 0.0,
    VI_Heat_Recovery_Enabled := L_Policy_Normal,
    VI_Is_Active := (VO_Supply_Fans[1] > 0) OR (VO_Exhaust_Fans[1] > 0),
    VI_Fan_Speed_Actual := BYTE_TO_REAL(VO_Supply_Fans[1]),
    VI_Supply_Temp := VI_Supply_Temps[1],
    VI_Extract_Temp := VI_Room_Temps[1],
    VI_Filter_Dirty := FALSE,
    VI_Alarm_Active := GVL_STATE.G_Ventilation_IO_Fault OR GVL_STATE.G_Ventilation_Subsystem_Degraded,
    VO_Command_Shadow => L_Vent_Command_Shadow,
    VO_State_Shadow => L_Vent_State_Shadow
);

// Ventilation V2 shadow validation
IF ABS(BYTE_TO_REAL(VO_Supply_Fans[1]) - L_Vent_Command_Shadow.Fan_Speed_Setpoint) > 0.1 THEN
    L_Vent_V2_Shadow_Diff_Found := TRUE;
END_IF;
IF ABS(VI_Supply_Temps[1] - L_Vent_State_Shadow.Supply_Temp) > 0.1 THEN
    L_Vent_V2_Shadow_Diff_Found := TRUE;
END_IF;

// Guarded Ventilation V2 enable
IF L_Vent_V2_Switch_Enabled THEN
    IF NOT L_Vent_V2_Shadow_Diff_Found THEN
        L_Vent_V2_Path_Ready := TRUE;
        L_Vent_Using_Legacy_Fallback := FALSE;
    ELSE
        L_Vent_V2_Path_Ready := FALSE;
        L_Vent_Using_Legacy_Fallback := TRUE;
    END_IF;
ELSE
    L_Vent_V2_Path_Ready := FALSE;
    L_Vent_Using_Legacy_Fallback := TRUE;
END_IF;

// 4. Формирование статусного сообщения
IF L_Policy_Safe_Stop THEN
    VO_Status_Msg := 'ВЕНТИЛЯЦИЯ: ОСТАНОВЛЕНА POLICY SAFE_STOP';
ELSIF L_Policy_Freeze_Protection THEN
    VO_Status_Msg := 'ВЕНТИЛЯЦИЯ: FREEZE_PROTECTION POLICY (stop)';
ELSIF L_Policy_Degraded THEN
    VO_Status_Msg := 'ВЕНТИЛЯЦИЯ: DEGRADED POLICY';
ELSE
    VO_Status_Msg := 'Вентиляция работает в штатном режиме';
END_IF;
// >>> BULK_SYNC_ANCHOR: FB_Ventilation_System_Manager <<<
    
END_FUNCTION_BLOCK

FUNCTION_BLOCK FB_Watchdog
  VAR_INPUT
    VI_System_Time_MS : UDINT;
    VI_Timeout_MS : UDINT := 2000;
  END_VAR
  VAR_OUTPUT
    VO_Alive : BOOL;
    VO_Watchdog_Fault : BOOL;
    VO_Cycle_DT_MS : UDINT;
  END_VAR
  VAR
    L_Initialized : BOOL := FALSE;
    L_Last_Call_MS : UDINT := 0;
    L_DT_MS : UDINT := 0;
  END_VAR

      IF NOT L_Initialized THEN
    L_Initialized := TRUE;
    L_Last_Call_MS := VI_System_Time_MS;
    VO_Cycle_DT_MS := 0;
    VO_Watchdog_Fault := FALSE;
    VO_Alive := TRUE;
    RETURN;
END_IF;

// Measure real time gap between successive calls
L_DT_MS := F_TimeDiff(VI_System_Time_MS, L_Last_Call_MS);
VO_Cycle_DT_MS := L_DT_MS;

// Fault if the task/cycle resumed after an abnormal pause
VO_Watchdog_Fault := (L_DT_MS > VI_Timeout_MS);
VO_Alive := NOT VO_Watchdog_Fault;

// Store current timestamp for next cycle
L_Last_Call_MS := VI_System_Time_MS;
// >>> BULK_SYNC_ANCHOR: FB_Watchdog <<<
    
END_FUNCTION_BLOCK

